  LIN {X -14931.996,Y 2667.355,Z 240.712,A 89.99946,B 0.00000,C 180.00000} ; retreat
  ; Step 2234, bar 855
  LIN {X -14831.996,Y 2667.355,Z 1143.930,A 89.99946,B 0.00000,C 180.00000} ; outside
  LIN {X -14831.996,Y 2667.355,Z 190.712,A 89.99946,B 0.00000,C 180.00000} ; preinsert
  LIN {X -14831.996,Y 2667.355,Z -59.288,A 89.99946,B 0.00000,C 180.00000} ; insert
  LIN {X -14831.996,Y 2667.355,Z -59.288,A 89.99946,B 0.00000,C 180.00000} ; release
  LIN {X -14831.996,Y 2667.355,Z 240.712,A 89.99946,B 0.00000,C 180.00000} ; retreat
  ; Step 2235, bar 853
  LIN {X -14731.996,Y 2667.355,Z 1143.930,A 89.99946,B 0.00000,C 180.00000} ; outside
  LIN {X -14731.996,Y 2667.355,Z 190.712,A 89.99946,B 0.00000,C 180.00000} ; preinsert
  LIN {X -14731.996,Y 2667.355,Z -59.288,A 89.99946,B 0.00000,C 180.00000} ; insert
  LIN {X -14731.996,Y 2667.355,Z -59.288,A 89.99946,B 0.00000,C 180.00000} ; release
  LIN {X -14731.996,Y 2667.355,Z 240.712,A 89.99946,B 0.00000,C 180.00000} ; retreat
  ; Step 2236, bar 851
  LIN {X -14631.996,Y 2667.355,Z 1143.930,A 89.99946,B 0.00000,C 180.00000} ; outside
  LIN {X -14631.996,Y 2667.355,Z 190.712,A 89.99946,B 0.00000,C 180.00000} ; preinsert
  LIN {X -14631.996,Y 2667.355,Z -59.288,A 89.99946,B 0.00000,C 180.00000} ; insert
  LIN {X -14631.996,Y 2667.355,Z -59.288,A 89.99946,B 0.00000,C 180.00000} ; release
  LIN {X -14631.996,Y 2667.355,Z 240.712,A 89.99946,B 0.00000,C 180.00000} ; retreat
  ; Step 2237, bar 849
  LIN {X -14531.996,Y 2667.355,Z 1143.930,A 89.99946,B 0.00000,C 180.00000} ; outside
  LIN {X -14531.996,Y 2667.355,Z 190.712,A 89.99946,B 0.00000,C 180.00000} ; preinsert
  LIN {X -14531.996,Y 2667.355,Z -59.288,A 89.99946,B 0.00000,C 180.00000} ; insert
  LIN {X -14531.996,Y 2667.355,Z -59.288,A 89.99946,B 0.00000,C 180.00000} ; release
  LIN {X -14531.996,Y 2667.355,Z 240.712,A 89.99946,B 0.00000,C 180.00000} ; retreat
  ; Step 2238, bar 847
  LIN {X -14431.996,Y 2667.355,Z 1143.930,A 89.99946,B 0.00000,C 180.00000} ; outside
  LIN {X -14431.996,Y 2667.355,Z 190.712,A 89.99946,B 0.00000,C 180.00000} ; preinsert
  LIN {X -14431.996,Y 2667.355,Z -59.288,A 89.99946,B 0.00000,C 180.00000} ; insert
  LIN {X -14431.996,Y 2667.355,Z -59.288,A 89.99946,B 0.00000,C 180.00000} ; release
  LIN {X -14431.996,Y 2667.355,Z 240.712,A 89.99946,B 0.00000,C 180.00000} ; retreat
  ; Step 2239, bar 845
  LIN {X -14331.996,Y 2667.355,Z 1143.930,A 89.99946,B 0.00000,C 180.00000} ; outside
  LIN {X -14331.996,Y 2667.355,Z 190.712,A 89.99946,B 0.00000,C 180.00000} ; preinsert
  LIN {X -14331.996,Y 2667.355,Z -59.288,A 89.99946,B 0.00000,C 180.00000} ; insert
  LIN {X -14331.996,Y 2667.355,Z -59.288,A 89.99946,B 0.00000,C 180.00000} ; release
  LIN {X -14331.996,Y 2667.355,Z 240.712,A 89.99946,B 0.00000,C 180.00000} ; retreat
  ; Step 2240, bar 843
  LIN {X -14231.996,Y 2667.355,Z 1143.930,A 89.99946,B 0.00000,C 180.00000} ; outside
  LIN {X -14231.996,Y 2667.355,Z 190.712,A 89.99946,B 0.00000,C 180.00000} ; preinsert
  LIN {X -14231.996,Y 2667.355,Z -59.288,A 89.99946,B 0.00000,C 180.00000} ; insert
  LIN {X -14231.996,Y 2667.355,Z -59.288,A 89.99946,B 0.00000,C 180.00000} ; release
  LIN {X -14231.996,Y 2667.355,Z 240.712,A 89.99946,B 0.00000,C 180.00000} ; retreat
  ; Step 2241, bar 841
  LIN {X -14131.996,Y 2667.355,Z 1143.930,A 89.99946,B 0.00000,C 180.00000} ; outside
  LIN {X -14131.996,Y 2667.355,Z 190.712,A 89.99946,B 0.00000,C 180.00000} ; preinsert
  LIN {X -14131.996,Y 2667.355,Z -59.288,A 89.99946,B 0.00000,C 180.00000} ; insert
  LIN {X -14131.996,Y 2667.355,Z -59.288,A 89.99946,B 0.00000,C 180.00000} ; release
  LIN {X -14131.996,Y 2667.355,Z 240.712,A 89.99946,B 0.00000,C 180.00000} ; retreat
  ; Step 2242, bar 839
  LIN {X -13831.996,Y 2667.355,Z 1143.930,A 89.99946,B 0.00000,C 180.00000} ; outside
  LIN {X -13831.996,Y 2667.355,Z 190.712,A 89.99946,B 0.00000,C 180.00000} ; preinsert
  LIN {X -13831.996,Y 2667.355,Z -59.288,A 89.99946,B 0.00000,C 180.00000} ; insert
  LIN {X -13831.996,Y 2667.355,Z -59.288,A 89.99946,B 0.00000,C 180.00000} ; release
  LIN {X -13831.996,Y 2667.355,Z 240.712,A 89.99946,B 0.00000,C 180.00000} ; retreat
  ; Step 2243, bar 837
  LIN {X -13731.996,Y 2667.355,Z 1143.930,A 89.99946,B 0.00000,C 180.00000} ; outside
  LIN {X -13731.996,Y 2667.355,Z 190.712,A 89.99946,B 0.00000,C 180.00000} ; preinsert
  LIN {X -13731.996,Y 2667.355,Z -59.288,A 89.99946,B 0.00000,C 180.00000} ; insert
  LIN {X -13731.996,Y 2667.355,Z -59.288,A 89.99946,B 0.00000,C 180.00000} ; release
  LIN {X -13731.996,Y 2667.355,Z 240.712,A 89.99946,B 0.00000,C 180.00000} ; retreat
  ; Step 2244, bar 835
  LIN {X -13631.996,Y 2667.355,Z 1143.930,A 89.99946,B 0.00000,C 180.00000} ; outside
  LIN {X -13631.996,Y 2667.355,Z 190.712,A 89.99946,B 0.00000,C 180.00000} ; preinsert
  LIN {X -13631.996,Y 2667.355,Z -59.288,A 89.99946,B 0.00000,C 180.00000} ; insert
  LIN {X -13631.996,Y 2667.355,Z -59.288,A 89.99946,B 0.00000,C 180.00000} ; release
  LIN {X -13631.996,Y 2667.355,Z 240.712,A 89.99946,B 0.00000,C 180.00000} ; retreat
  ; Step 2245, bar 833
  LIN {X -13531.996,Y 2667.355,Z 1143.930,A 89.99946,B 0.00000,C 180.00000} ; outside
  LIN {X -13531.996,Y 2667.355,Z 190.712,A 89.99946,B 0.00000,C 180.00000} ; preinsert
  LIN {X -13531.996,Y 2667.355,Z -59.288,A 89.99946,B 0.00000,C 180.00000} ; insert
  LIN {X -13531.996,Y 2667.355,Z -59.288,A 89.99946,B 0.00000,C 180.00000} ; release
  LIN {X -13531.996,Y 2667.355,Z 240.712,A 89.99946,B 0.00000,C 180.00000} ; retreat
  ; Step 2246, bar 831
  LIN {X -13431.996,Y 2667.355,Z 1143.930,A 89.99946,B 0.00000,C 180.00000} ; outside
  LIN {X -13431.996,Y 2667.355,Z 190.712,A 89.99946,B 0.00000,C 180.00000} ; preinsert
  LIN {X -13431.996,Y 2667.355,Z -59.288,A 89.99946,B 0.00000,C 180.00000} ; insert
  LIN {X -13431.996,Y 2667.355,Z -59.288,A 89.99946,B 0.00000,C 180.00000} ; release
  LIN {X -13431.996,Y 2667.355,Z 240.712,A 89.99946,B 0.00000,C 180.00000} ; retreat
  ; Step 2247, bar 829
  LIN {X -13331.996,Y 2667.355,Z 1143.930,A 89.99946,B 0.00000,C 180.00000} ; outside
  LIN {X -13331.996,Y 2667.355,Z 190.712,A 89.99946,B 0.00000,C 180.00000} ; preinsert
  LIN {X -13331.996,Y 2667.355,Z -59.288,A 89.99946,B 0.00000,C 180.00000} ; insert
  LIN {X -13331.996,Y 2667.355,Z -59.288,A 89.99946,B 0.00000,C 180.00000} ; release
  LIN {X -13331.996,Y 2667.355,Z 240.712,A 89.99946,B 0.00000,C 180.00000} ; retreat
  ; Step 2248, bar 827
  LIN {X -13231.996,Y 2667.355,Z 1143.930,A 89.99946,B 0.00000,C 180.00000} ; outside
  LIN {X -13231.996,Y 2667.355,Z 190.712,A 89.99946,B 0.00000,C 180.00000} ; preinsert
  LIN {X -13231.996,Y 2667.355,Z -59.288,A 89.99946,B 0.00000,C 180.00000} ; insert
  LIN {X -13231.996,Y 2667.355,Z -59.288,A 89.99946,B 0.00000,C 180.00000} ; release
  LIN {X -13231.996,Y 2667.355,Z 240.712,A 89.99946,B 0.00000,C 180.00000} ; retreat
  ; Step 2249, bar 825
  LIN {X -13131.996,Y 2667.355,Z 1143.930,A 89.99946,B 0.00000,C 180.00000} ; outside
  LIN {X -13131.996,Y 2667.355,Z 190.712,A 89.99946,B 0.00000,C 180.00000} ; preinsert
  LIN {X -13131.996,Y 2667.355,Z -59.288,A 89.99946,B 0.00000,C 180.00000} ; insert
  LIN {X -13131.996,Y 2667.355,Z -59.288,A 89.99946,B 0.00000,C 180.00000} ; release
  LIN {X -13131.996,Y 2667.355,Z 240.712,A 89.99946,B 0.00000,C 180.00000} ; retreat
  ; Step 2250, bar 823
  LIN {X -13031.996,Y 2667.355,Z 1143.930,A 89.99946,B 0.00000,C 180.00000} ; outside
  LIN {X -13031.996,Y 2667.355,Z 190.712,A 89.99946,B 0.00000,C 180.00000} ; preinsert
  LIN {X -13031.996,Y 2667.355,Z -59.288,A 89.99946,B 0.00000,C 180.00000} ; insert
  LIN {X -13031.996,Y 2667.355,Z -59.288,A 89.99946,B 0.00000,C 180.00000} ; release
  LIN {X -13031.996,Y 2667.355,Z 240.712,A 89.99946,B 0.00000,C 180.00000} ; retreat
  ; Step 2251, bar 821
  LIN {X -12931.996,Y 2667.355,Z 1143.930,A 89.99946,B 0.00000,C 180.00000} ; outside
  LIN {X -12931.996,Y 2667.355,Z 190.712,A 89.99946,B 0.00000,C 180.00000} ; preinsert
  LIN {X -12931.996,Y 2667.355,Z -59.288,A 89.99946,B 0.00000,C 180.00000} ; insert
  LIN {X -12931.996,Y 2667.355,Z -59.288,A 89.99946,B 0.00000,C 180.00000} ; release
  LIN {X -12931.996,Y 2667.355,Z 240.712,A 89.99946,B 0.00000,C 180.00000} ; retreat
  ; Step 2252, bar 819
  LIN {X -12831.996,Y 2667.355,Z 1143.930,A 89.99946,B 0.00000,C 180.00000} ; outside
  LIN {X -12831.996,Y 2667.355,Z 190.712,A 89.99946,B 0.00000,C 180.00000} ; preinsert
  LIN {X -12831.996,Y 2667.355,Z -59.288,A 89.99946,B 0.00000,C 180.00000} ; insert
  LIN {X -12831.996,Y 2667.355,Z -59.288,A 89.99946,B 0.00000,C 180.00000} ; release
  LIN {X -12831.996,Y 2667.355,Z 240.712,A 89.99946,B 0.00000,C 180.00000} ; retreat
  ; Step 2253, bar 817
  LIN {X -12731.996,Y 2667.355,Z 1143.930,A 89.99946,B 0.00000,C 180.00000} ; outside
  LIN {X -12731.996,Y 2667.355,Z 190.712,A 89.99946,B 0.00000,C 180.00000} ; preinsert
  LIN {X -12731.996,Y 2667.355,Z -59.288,A 89.99946,B 0.00000,C 180.00000} ; insert
  LIN {X -12731.996,Y 2667.355,Z -59.288,A 89.99946,B 0.00000,C 180.00000} ; release
  LIN {X -12731.996,Y 2667.355,Z 240.712,A 89.99946,B 0.00000,C 180.00000} ; retreat
  ; Step 2254, bar 815
  LIN {X -12631.996,Y 2667.355,Z 1143.930,A 89.99946,B 0.00000,C 180.00000} ; outside
  LIN {X -12631.996,Y 2667.355,Z 190.712,A 89.99946,B 0.00000,C 180.00000} ; preinsert
  LIN {X -12631.996,Y 2667.355,Z -59.288,A 89.99946,B 0.00000,C 180.00000} ; insert
  LIN {X -12631.996,Y 2667.355,Z -59.288,A 89.99946,B 0.00000,C 180.00000} ; release
  LIN {X -12631.996,Y 2667.355,Z 240.712,A 89.99946,B 0.00000,C 180.00000} ; retreat
  ; Step 2255, bar 813
  LIN {X -12531.996,Y 2667.355,Z 1143.930,A 89.99946,B 0.00000,C 180.00000} ; outside
  LIN {X -12531.996,Y 2667.355,Z 190.712,A 89.99946,B 0.00000,C 180.00000} ; preinsert
  LIN {X -12531.996,Y 2667.355,Z -59.288,A 89.99946,B 0.00000,C 180.00000} ; insert
  LIN {X -12531.996,Y 2667.355,Z -59.288,A 89.99946,B 0.00000,C 180.00000} ; release
  LIN {X -12531.996,Y 2667.355,Z 240.712,A 89.99946,B 0.00000,C 180.00000} ; retreat
  ; Step 2256, bar 811
  LIN {X -12431.996,Y 2667.355,Z 1143.930,A 89.99946,B 0.00000,C 180.00000} ; outside
  LIN {X -12431.996,Y 2667.355,Z 190.712,A 89.99946,B 0.00000,C 180.00000} ; preinsert
  LIN {X -12431.996,Y 2667.355,Z -59.288,A 89.99946,B 0.00000,C 180.00000} ; insert
  LIN {X -12431.996,Y 2667.355,Z -59.288,A 89.99946,B 0.00000,C 180.00000} ; release
  LIN {X -12431.996,Y 2667.355,Z 240.712,A 89.99946,B 0.00000,C 180.00000} ; retreat
  ; Step 2257, bar 809
  LIN {X -12331.996,Y 2667.355,Z 1143.930,A 89.99946,B 0.00000,C 180.00000} ; outside
  LIN {X -12331.996,Y 2667.355,Z 190.712,A 89.99946,B 0.00000,C 180.00000} ; preinsert
  LIN {X -12331.996,Y 2667.355,Z -59.288,A 89.99946,B 0.00000,C 180.00000} ; insert
  LIN {X -12331.996,Y 2667.355,Z -59.288,A 89.99946,B 0.00000,C 180.00000} ; release
  LIN {X -12331.996,Y 2667.355,Z 240.712,A 89.99946,B 0.00000,C 180.00000} ; retreat
  ; Step 2258, bar 807
  LIN {X -12231.996,Y 2667.355,Z 1143.930,A 89.99946,B 0.00000,C 180.00000} ; outside
  LIN {X -12231.996,Y 2667.355,Z 190.712,A 89.99946,B 0.00000,C 180.00000} ; preinsert
  LIN {X -12231.996,Y 2667.355,Z -59.288,A 89.99946,B 0.00000,C 180.00000} ; insert
  LIN {X -12231.996,Y 2667.355,Z -59.288,A 89.99946,B 0.00000,C 180.00000} ; release
  LIN {X -12231.996,Y 2667.355,Z 240.712,A 89.99946,B 0.00000,C 180.00000} ; retreat
  ; Step 2259, bar 805
  LIN {X -12106.996,Y 2667.355,Z 1143.930,A 89.99946,B 0.00000,C 180.00000} ; outside
  LIN {X -12106.996,Y 2667.355,Z 190.712,A 89.99946,B 0.00000,C 180.00000} ; preinsert
  LIN {X -12106.996,Y 2667.355,Z -59.288,A 89.99946,B 0.00000,C 180.00000} ; insert
  LIN {X -12106.996,Y 2667.355,Z -59.288,A 89.99946,B 0.00000,C 180.00000} ; release
  LIN {X -12106.996,Y 2667.355,Z 240.712,A 89.99946,B 0.00000,C 180.00000} ; retreat
  ; Step 2260, bar 803
  LIN {X -11981.996,Y 2667.355,Z 1143.930,A 89.99946,B 0.00000,C 180.00000} ; outside
  LIN {X -11981.996,Y 2667.355,Z 190.712,A 89.99946,B 0.00000,C 180.00000} ; preinsert
  LIN {X -11981.996,Y 2667.355,Z -59.288,A 89.99946,B 0.00000,C 180.00000} ; insert
  LIN {X -11981.996,Y 2667.355,Z -59.288,A 89.99946,B 0.00000,C 180.00000} ; release
  LIN {X -11981.996,Y 2667.355,Z 240.712,A 89.99946,B 0.00000,C 180.00000} ; retreat
  ; Step 2261, bar 801
  LIN {X -11856.996,Y 2667.355,Z 1143.930,A 89.99946,B 0.00000,C 180.00000} ; outside
  LIN {X -11856.996,Y 2667.355,Z 190.712,A 89.99946,B 0.00000,C 180.00000} ; preinsert
  LIN {X -11856.996,Y 2667.355,Z -59.288,A 89.99946,B 0.00000,C 180.00000} ; insert
  LIN {X -11856.996,Y 2667.355,Z -59.288,A 89.99946,B 0.00000,C 180.00000} ; release
  LIN {X -11856.996,Y 2667.355,Z 240.712,A 89.99946,B 0.00000,C 180.00000} ; retreat
  ; Step 2262, bar 799
  LIN {X -11731.996,Y 2667.355,Z 1143.930,A 89.99946,B 0.00000,C 180.00000} ; outside
  LIN {X -11731.996,Y 2667.355,Z 190.712,A 89.99946,B 0.00000,C 180.00000} ; preinsert
  LIN {X -11731.996,Y 2667.355,Z -59.288,A 89.99946,B 0.00000,C 180.00000} ; insert
  LIN {X -11731.996,Y 2667.355,Z -59.288,A 89.99946,B 0.00000,C 180.00000} ; release
  LIN {X -11731.996,Y 2667.355,Z 240.712,A 89.99946,B 0.00000,C 180.00000} ; retreat
  ; Step 2263, bar 797
  LIN {X -11606.996,Y 2667.355,Z 1143.930,A 89.99946,B 0.00000,C 180.00000} ; outside
  LIN {X -11606.996,Y 2667.355,Z 190.712,A 89.99946,B 0.00000,C 180.00000} ; preinsert
  LIN {X -11606.996,Y 2667.355,Z -59.288,A 89.99946,B 0.00000,C 180.00000} ; insert
  LIN {X -11606.996,Y 2667.355,Z -59.288,A 89.99946,B 0.00000,C 180.00000} ; release
  LIN {X -11606.996,Y 2667.355,Z 240.712,A 89.99946,B 0.00000,C 180.00000} ; retreat
  ; Step 2264, bar 795
  LIN {X -11481.996,Y 2667.355,Z 1143.930,A 89.99946,B 0.00000,C 180.00000} ; outside
  LIN {X -11481.996,Y 2667.355,Z 190.712,A 89.99946,B 0.00000,C 180.00000} ; preinsert
  LIN {X -11481.996,Y 2667.355,Z -59.288,A 89.99946,B 0.00000,C 180.00000} ; insert
  LIN {X -11481.996,Y 2667.355,Z -59.288,A 89.99946,B 0.00000,C 180.00000} ; release
  LIN {X -11481.996,Y 2667.355,Z 240.712,A 89.99946,B 0.00000,C 180.00000} ; retreat
  ; Step 2265, bar 793
  LIN {X -11356.996,Y 2667.355,Z 1143.930,A 89.99946,B 0.00000,C 180.00000} ; outside
  LIN {X -11356.996,Y 2667.355,Z 190.712,A 89.99946,B 0.00000,C 180.00000} ; preinsert
  LIN {X -11356.996,Y 2667.355,Z -59.288,A 89.99946,B 0.00000,C 180.00000} ; insert
  LIN {X -11356.996,Y 2667.355,Z -59.288,A 89.99946,B 0.00000,C 180.00000} ; release
  LIN {X -11356.996,Y 2667.355,Z 240.712,A 89.99946,B 0.00000,C 180.00000} ; retreat
  ; Step 2266, bar 791
  LIN {X -11231.996,Y 2667.355,Z 1143.930,A 89.99946,B 0.00000,C 180.00000} ; outside
  LIN {X -11231.996,Y 2667.355,Z 190.712,A 89.99946,B 0.00000,C 180.00000} ; preinsert
  LIN {X -11231.996,Y 2667.355,Z -59.288,A 89.99946,B 0.00000,C 180.00000} ; insert
  LIN {X -11231.996,Y 2667.355,Z -59.288,A 89.99946,B 0.00000,C 180.00000} ; release
  LIN {X -11231.996,Y 2667.355,Z 240.712,A 89.99946,B 0.00000,C 180.00000} ; retreat
  ; Step 2267, bar 789
  LIN {X -11106.996,Y 2667.355,Z 1143.930,A 89.99946,B 0.00000,C 180.00000} ; outside
  LIN {X -11106.996,Y 2667.355,Z 190.712,A 89.99946,B 0.00000,C 180.00000} ; preinsert
  LIN {X -11106.996,Y 2667.355,Z -59.288,A 89.99946,B 0.00000,C 180.00000} ; insert
  LIN {X -11106.996,Y 2667.355,Z -59.288,A 89.99946,B 0.00000,C 180.00000} ; release
  LIN {X -11106.996,Y 2667.355,Z 240.712,A 89.99946,B 0.00000,C 180.00000} ; retreat
  ; Step 2268, bar 787
  LIN {X -10981.996,Y 2667.355,Z 1143.930,A 89.99946,B 0.00000,C 180.00000} ; outside
  LIN {X -10981.996,Y 2667.355,Z 190.712,A 89.99946,B 0.00000,C 180.00000} ; preinsert
  LIN {X -10981.996,Y 2667.355,Z -59.288,A 89.99946,B 0.00000,C 180.00000} ; insert
  LIN {X -10981.996,Y 2667.355,Z -59.288,A 89.99946,B 0.00000,C 180.00000} ; release
  LIN {X -10981.996,Y 2667.355,Z 240.712,A 89.99946,B 0.00000,C 180.00000} ; retreat
  ; Step 2269, bar 785
  LIN {X -10856.996,Y 2667.355,Z 1143.930,A 89.99946,B 0.00000,C 180.00000} ; outside
  LIN {X -10856.996,Y 2667.355,Z 190.712,A 89.99946,B 0.00000,C 180.00000} ; preinsert
  LIN {X -10856.996,Y 2667.355,Z -59.288,A 89.99946,B 0.00000,C 180.00000} ; insert
  LIN {X -10856.996,Y 2667.355,Z -59.288,A 89.99946,B 0.00000,C 180.00000} ; release
  LIN {X -10856.996,Y 2667.355,Z 240.712,A 89.99946,B 0.00000,C 180.00000} ; retreat
  ; Step 2270, bar 783
  LIN {X -10731.996,Y 2667.355,Z 1143.930,A 89.99946,B 0.00000,C 180.00000} ; outside
  LIN {X -10731.996,Y 2667.355,Z 190.712,A 89.99946,B 0.00000,C 180.00000} ; preinsert
  LIN {X -10731.996,Y 2667.355,Z -59.288,A 89.99946,B 0.00000,C 180.00000} ; insert
  LIN {X -10731.996,Y 2667.355,Z -59.288,A 89.99946,B 0.00000,C 180.00000} ; release
  LIN {X -10731.996,Y 2667.355,Z 240.712,A 89.99946,B 0.00000,C 180.00000} ; retreat
  ; Step 2271, bar 781
  LIN {X -10606.996,Y 2667.355,Z 1143.930,A 89.99946,B 0.00000,C 180.00000} ; outside
  LIN {X -10606.996,Y 2667.355,Z 190.712,A 89.99946,B 0.00000,C 180.00000} ; preinsert
  LIN {X -10606.996,Y 2667.355,Z -59.288,A 89.99946,B 0.00000,C 180.00000} ; insert
  LIN {X -10606.996,Y 2667.355,Z -59.288,A 89.99946,B 0.00000,C 180.00000} ; release
  LIN {X -10606.996,Y 2667.355,Z 240.712,A 89.99946,B 0.00000,C 180.00000} ; retreat
  ; Step 2272, bar 779
  LIN {X -10481.996,Y 2667.355,Z 1143.930,A 89.99946,B 0.00000,C 180.00000} ; outside
  LIN {X -10481.996,Y 2667.355,Z 190.712,A 89.99946,B 0.00000,C 180.00000} ; preinsert
  LIN {X -10481.996,Y 2667.355,Z -59.288,A 89.99946,B 0.00000,C 180.00000} ; insert
  LIN {X -10481.996,Y 2667.355,Z -59.288,A 89.99946,B 0.00000,C 180.00000} ; release
  LIN {X -10481.996,Y 2667.355,Z 240.712,A 89.99946,B 0.00000,C 180.00000} ; retreat
  ; Step 2273, bar 777
  LIN {X -10356.996,Y 2667.355,Z 1143.930,A 89.99946,B 0.00000,C 180.00000} ; outside
  LIN {X -10356.996,Y 2667.355,Z 190.712,A 89.99946,B 0.00000,C 180.00000} ; preinsert
  LIN {X -10356.996,Y 2667.355,Z -59.288,A 89.99946,B 0.00000,C 180.00000} ; insert
  LIN {X -10356.996,Y 2667.355,Z -59.288,A 89.99946,B 0.00000,C 180.00000} ; release
  LIN {X -10356.996,Y 2667.355,Z 240.712,A 89.99946,B 0.00000,C 180.00000} ; retreat
  ; Step 2274, bar 775
  LIN {X -10231.996,Y 2667.355,Z 1143.930,A 89.99946,B 0.00000,C 180.00000} ; outside
  LIN {X -10231.996,Y 2667.355,Z 190.712,A 89.99946,B 0.00000,C 180.00000} ; preinsert
  LIN {X -10231.996,Y 2667.355,Z -59.288,A 89.99946,B 0.00000,C 180.00000} ; insert
  LIN {X -10231.996,Y 2667.355,Z -59.288,A 89.99946,B 0.00000,C 180.00000} ; release
  LIN {X -10231.996,Y 2667.355,Z 240.712,A 89.99946,B 0.00000,C 180.00000} ; retreat
  ; Step 2275, bar 773
  LIN {X -10106.996,Y 2667.355,Z 1143.930,A 89.99946,B 0.00000,C 180.00000} ; outside
  LIN {X -10106.996,Y 2667.355,Z 190.712,A 89.99946,B 0.00000,C 180.00000} ; preinsert
  LIN {X -10106.996,Y 2667.355,Z -59.288,A 89.99946,B 0.00000,C 180.00000} ; insert
  LIN {X -10106.996,Y 2667.355,Z -59.288,A 89.99946,B 0.00000,C 180.00000} ; release
  LIN {X -10106.996,Y 2667.355,Z 240.712,A 89.99946,B 0.00000,C 180.00000} ; retreat
  ; Step 2276, bar 771
  LIN {X -9856.996,Y 2667.355,Z 1143.930,A 89.99946,B 0.00000,C 180.00000} ; outside
  LIN {X -9856.996,Y 2667.355,Z 190.712,A 89.99946,B 0.00000,C 180.00000} ; preinsert
  LIN {X -9856.996,Y 2667.355,Z -59.288,A 89.99946,B 0.00000,C 180.00000} ; insert
  LIN {X -9856.996,Y 2667.355,Z -59.288,A 89.99946,B 0.00000,C 180.00000} ; release
  LIN {X -9856.996,Y 2667.355,Z 240.712,A 89.99946,B 0.00000,C 180.00000} ; retreat
  ; Step 2277, bar 769
  LIN {X -9731.996,Y 2667.355,Z 1143.930,A 89.99946,B 0.00000,C 180.00000} ; outside
  LIN {X -9731.996,Y 2667.355,Z 190.712,A 89.99946,B 0.00000,C 180.00000} ; preinsert
  LIN {X -9731.996,Y 2667.355,Z -59.288,A 89.99946,B 0.00000,C 180.00000} ; insert
  LIN {X -9731.996,Y 2667.355,Z -59.288,A 89.99946,B 0.00000,C 180.00000} ; release
  LIN {X -9731.996,Y 2667.355,Z 240.712,A 89.99946,B 0.00000,C 180.00000} ; retreat
  ; Step 2278, bar 767
  LIN {X -9606.996,Y 2667.355,Z 1143.930,A 89.99946,B 0.00000,C 180.00000} ; outside
  LIN {X -9606.996,Y 2667.355,Z 190.712,A 89.99946,B 0.00000,C 180.00000} ; preinsert
  LIN {X -9606.996,Y 2667.355,Z -59.288,A 89.99946,B 0.00000,C 180.00000} ; insert
  LIN {X -9606.996,Y 2667.355,Z -59.288,A 89.99946,B 0.00000,C 180.00000} ; release
  LIN {X -9606.996,Y 2667.355,Z 240.712,A 89.99946,B 0.00000,C 180.00000} ; retreat
  ; Step 2279, bar 765
  LIN {X -9481.996,Y 2667.355,Z 1143.930,A 89.99946,B 0.00000,C 180.00000} ; outside
  LIN {X -9481.996,Y 2667.355,Z 190.712,A 89.99946,B 0.00000,C 180.00000} ; preinsert
  LIN {X -9481.996,Y 2667.355,Z -59.288,A 89.99946,B 0.00000,C 180.00000} ; insert
  LIN {X -9481.996,Y 2667.355,Z -59.288,A 89.99946,B 0.00000,C 180.00000} ; release
  LIN {X -9481.996,Y 2667.355,Z 240.712,A 89.99946,B 0.00000,C 180.00000} ; retreat
  ; Step 2280, bar 763
  LIN {X -9356.996,Y 2667.355,Z 1143.930,A 89.99946,B 0.00000,C 180.00000} ; outside
  LIN {X -9356.996,Y 2667.355,Z 190.712,A 89.99946,B 0.00000,C 180.00000} ; preinsert
  LIN {X -9356.996,Y 2667.355,Z -59.288,A 89.99946,B 0.00000,C 180.00000} ; insert
  LIN {X -9356.996,Y 2667.355,Z -59.288,A 89.99946,B 0.00000,C 180.00000} ; release
  LIN {X -9356.996,Y 2667.355,Z 240.712,A 89.99946,B 0.00000,C 180.00000} ; retreat
  ; Step 2281, bar 761
  LIN {X -9231.996,Y 2667.355,Z 1143.930,A 89.99946,B 0.00000,C 180.00000} ; outside
  LIN {X -9231.996,Y 2667.355,Z 190.712,A 89.99946,B 0.00000,C 180.00000} ; preinsert
  LIN {X -9231.996,Y 2667.355,Z -59.288,A 89.99946,B 0.00000,C 180.00000} ; insert
  LIN {X -9231.996,Y 2667.355,Z -59.288,A 89.99946,B 0.00000,C 180.00000} ; release
  LIN {X -9231.996,Y 2667.355,Z 240.712,A 89.99946,B 0.00000,C 180.00000} ; retreat
  ; Step 2282, bar 759
  LIN {X -9106.996,Y 2667.355,Z 1143.930,A 89.99946,B 0.00000,C 180.00000} ; outside
  LIN {X -9106.996,Y 2667.355,Z 190.712,A 89.99946,B 0.00000,C 180.00000} ; preinsert
  LIN {X -9106.996,Y 2667.355,Z -59.288,A 89.99946,B 0.00000,C 180.00000} ; insert
  LIN {X -9106.996,Y 2667.355,Z -59.288,A 89.99946,B 0.00000,C 180.00000} ; release
  LIN {X -9106.996,Y 2667.355,Z 240.712,A 89.99946,B 0.00000,C 180.00000} ; retreat
  ; Step 2283, bar 757
  LIN {X -8981.996,Y 2667.355,Z 1143.930,A 89.99946,B 0.00000,C 180.00000} ; outside
  LIN {X -8981.996,Y 2667.355,Z 190.712,A 89.99946,B 0.00000,C 180.00000} ; preinsert
  LIN {X -8981.996,Y 2667.355,Z -59.288,A 89.99946,B 0.00000,C 180.00000} ; insert
  LIN {X -8981.996,Y 2667.355,Z -59.288,A 89.99946,B 0.00000,C 180.00000} ; release
  LIN {X -8981.996,Y 2667.355,Z 240.712,A 89.99946,B 0.00000,C 180.00000} ; retreat
  ; Step 2284, bar 755
  LIN {X -8856.996,Y 2667.355,Z 1143.930,A 89.99946,B 0.00000,C 180.00000} ; outside
  LIN {X -8856.996,Y 2667.355,Z 190.712,A 89.99946,B 0.00000,C 180.00000} ; preinsert
  LIN {X -8856.996,Y 2667.355,Z -59.288,A 89.99946,B 0.00000,C 180.00000} ; insert
  LIN {X -8856.996,Y 2667.355,Z -59.288,A 89.99946,B 0.00000,C 180.00000} ; release
  LIN {X -8856.996,Y 2667.355,Z 240.712,A 89.99946,B 0.00000,C 180.00000} ; retreat
  ; Step 2285, bar 753
  LIN {X -8731.996,Y 2667.355,Z 1143.930,A 89.99946,B 0.00000,C 180.00000} ; outside
  LIN {X -8731.996,Y 2667.355,Z 190.712,A 89.99946,B 0.00000,C 180.00000} ; preinsert
  LIN {X -8731.996,Y 2667.355,Z -59.288,A 89.99946,B 0.00000,C 180.00000} ; insert
  LIN {X -8731.996,Y 2667.355,Z -59.288,A 89.99946,B 0.00000,C 180.00000} ; release
  LIN {X -8731.996,Y 2667.355,Z 240.712,A 89.99946,B 0.00000,C 180.00000} ; retreat
  ; Step 2286, bar 751
  LIN {X -8606.996,Y 2667.355,Z 1143.930,A 89.99946,B 0.00000,C 180.00000} ; outside
  LIN {X -8606.996,Y 2667.355,Z 190.712,A 89.99946,B 0.00000,C 180.00000} ; preinsert
  LIN {X -8606.996,Y 2667.355,Z -59.288,A 89.99946,B 0.00000,C 180.00000} ; insert
  LIN {X -8606.996,Y 2667.355,Z -59.288,A 89.99946,B 0.00000,C 180.00000} ; release
  LIN {X -8606.996,Y 2667.355,Z 240.712,A 89.99946,B 0.00000,C 180.00000} ; retreat
  ; Step 2287, bar 749
  LIN {X -8481.996,Y 2667.355,Z 1143.930,A 89.99946,B 0.00000,C 180.00000} ; outside
  LIN {X -8481.996,Y 2667.355,Z 190.712,A 89.99946,B 0.00000,C 180.00000} ; preinsert
  LIN {X -8481.996,Y 2667.355,Z -59.288,A 89.99946,B 0.00000,C 180.00000} ; insert
  LIN {X -8481.996,Y 2667.355,Z -59.288,A 89.99946,B 0.00000,C 180.00000} ; release
  LIN {X -8481.996,Y 2667.355,Z 240.712,A 89.99946,B 0.00000,C 180.00000} ; retreat
  ; Step 2288, bar 747
  LIN {X -8356.996,Y 2667.355,Z 1143.930,A 89.99946,B 0.00000,C 180.00000} ; outside
  LIN {X -8356.996,Y 2667.355,Z 190.712,A 89.99946,B 0.00000,C 180.00000} ; preinsert
  LIN {X -8356.996,Y 2667.355,Z -59.288,A 89.99946,B 0.00000,C 180.00000} ; insert
  LIN {X -8356.996,Y 2667.355,Z -59.288,A 89.99946,B 0.00000,C 180.00000} ; release
  LIN {X -8356.996,Y 2667.355,Z 240.712,A 89.99946,B 0.00000,C 180.00000} ; retreat
  ; Step 2289, bar 745
  LIN {X -8231.996,Y 2667.355,Z 1143.930,A 89.99946,B 0.00000,C 180.00000} ; outside
  LIN {X -8231.996,Y 2667.355,Z 190.712,A 89.99946,B 0.00000,C 180.00000} ; preinsert
  LIN {X -8231.996,Y 2667.355,Z -59.288,A 89.99946,B 0.00000,C 180.00000} ; insert
  LIN {X -8231.996,Y 2667.355,Z -59.288,A 89.99946,B 0.00000,C 180.00000} ; release
  LIN {X -8231.996,Y 2667.355,Z 240.712,A 89.99946,B 0.00000,C 180.00000} ; retreat
  ; Step 2290, bar 743
  LIN {X -8106.996,Y 2667.355,Z 1143.930,A 89.99946,B 0.00000,C 180.00000} ; outside
  LIN {X -8106.996,Y 2667.355,Z 190.712,A 89.99946,B 0.00000,C 180.00000} ; preinsert
  LIN {X -8106.996,Y 2667.355,Z -59.288,A 89.99946,B 0.00000,C 180.00000} ; insert
  LIN {X -8106.996,Y 2667.355,Z -59.288,A 89.99946,B 0.00000,C 180.00000} ; release
  LIN {X -8106.996,Y 2667.355,Z 240.712,A 89.99946,B 0.00000,C 180.00000} ; retreat
  ; Step 2291, bar 741
  LIN {X -7981.996,Y 2667.355,Z 1143.930,A 89.99946,B 0.00000,C 180.00000} ; outside
  LIN {X -7981.996,Y 2667.355,Z 190.712,A 89.99946,B 0.00000,C 180.00000} ; preinsert
  LIN {X -7981.996,Y 2667.355,Z -59.288,A 89.99946,B 0.00000,C 180.00000} ; insert
  LIN {X -7981.996,Y 2667.355,Z -59.288,A 89.99946,B 0.00000,C 180.00000} ; release
  LIN {X -7981.996,Y 2667.355,Z 240.712,A 89.99946,B 0.00000,C 180.00000} ; retreat
  ; Step 2292, bar 739
  LIN {X -7856.996,Y 2667.355,Z 1143.930,A 89.99946,B 0.00000,C 180.00000} ; outside
  LIN {X -7856.996,Y 2667.355,Z 190.712,A 89.99946,B 0.00000,C 180.00000} ; preinsert
  LIN {X -7856.996,Y 2667.355,Z -59.288,A 89.99946,B 0.00000,C 180.00000} ; insert
  LIN {X -7856.996,Y 2667.355,Z -59.288,A 89.99946,B 0.00000,C 180.00000} ; release
  LIN {X -7856.996,Y 2667.355,Z 240.712,A 89.99946,B 0.00000,C 180.00000} ; retreat
  ; Step 2293, bar 737
  LIN {X -7731.996,Y 2667.355,Z 1143.930,A 89.99946,B 0.00000,C 180.00000} ; outside
  LIN {X -7731.996,Y 2667.355,Z 190.712,A 89.99946,B 0.00000,C 180.00000} ; preinsert
  LIN {X -7731.996,Y 2667.355,Z -59.288,A 89.99946,B 0.00000,C 180.00000} ; insert
  LIN {X -7731.996,Y 2667.355,Z -59.288,A 89.99946,B 0.00000,C 180.00000} ; release
  LIN {X -7731.996,Y 2667.355,Z 240.712,A 89.99946,B 0.00000,C 180.00000} ; retreat
  ; Step 2294, bar 735
  LIN {X -7606.996,Y 2667.355,Z 1143.930,A 89.99946,B 0.00000,C 180.00000} ; outside
  LIN {X -7606.996,Y 2667.355,Z 190.712,A 89.99946,B 0.00000,C 180.00000} ; preinsert
  LIN {X -7606.996,Y 2667.355,Z -59.288,A 89.99946,B 0.00000,C 180.00000} ; insert
  LIN {X -7606.996,Y 2667.355,Z -59.288,A 89.99946,B 0.00000,C 180.00000} ; release
  LIN {X -7606.996,Y 2667.355,Z 240.712,A 89.99946,B 0.00000,C 180.00000} ; retreat
  ; Step 2295, bar 733
  LIN {X -7481.996,Y 2667.355,Z 1143.930,A 89.99946,B 0.00000,C 180.00000} ; outside
  LIN {X -7481.996,Y 2667.355,Z 190.712,A 89.99946,B 0.00000,C 180.00000} ; preinsert
  LIN {X -7481.996,Y 2667.355,Z -59.288,A 89.99946,B 0.00000,C 180.00000} ; insert
  LIN {X -7481.996,Y 2667.355,Z -59.288,A 89.99946,B 0.00000,C 180.00000} ; release
  LIN {X -7481.996,Y 2667.355,Z 240.712,A 89.99946,B 0.00000,C 180.00000} ; retreat
  ; Step 2296, bar 731
  LIN {X -7356.996,Y 2667.355,Z 1143.930,A 89.99946,B 0.00000,C 180.00000} ; outside
  LIN {X -7356.996,Y 2667.355,Z 190.712,A 89.99946,B 0.00000,C 180.00000} ; preinsert
  LIN {X -7356.996,Y 2667.355,Z -59.288,A 89.99946,B 0.00000,C 180.00000} ; insert
  LIN {X -7356.996,Y 2667.355,Z -59.288,A 89.99946,B 0.00000,C 180.00000} ; release
  LIN {X -7356.996,Y 2667.355,Z 240.712,A 89.99946,B 0.00000,C 180.00000} ; retreat
  ; Step 2297, bar 729
  LIN {X -7231.996,Y 2667.355,Z 1143.930,A 89.99946,B 0.00000,C 180.00000} ; outside
  LIN {X -7231.996,Y 2667.355,Z 190.712,A 89.99946,B 0.00000,C 180.00000} ; preinsert
  LIN {X -7231.996,Y 2667.355,Z -59.288,A 89.99946,B 0.00000,C 180.00000} ; insert
  LIN {X -7231.996,Y 2667.355,Z -59.288,A 89.99946,B 0.00000,C 180.00000} ; release
  LIN {X -7231.996,Y 2667.355,Z 240.712,A 89.99946,B 0.00000,C 180.00000} ; retreat
  ; Step 2298, bar 727
  LIN {X -7106.996,Y 2667.355,Z 1143.930,A 89.99946,B 0.00000,C 180.00000} ; outside
  LIN {X -7106.996,Y 2667.355,Z 190.712,A 89.99946,B 0.00000,C 180.00000} ; preinsert
  LIN {X -7106.996,Y 2667.355,Z -59.288,A 89.99946,B 0.00000,C 180.00000} ; insert
  LIN {X -7106.996,Y 2667.355,Z -59.288,A 89.99946,B 0.00000,C 180.00000} ; release
  LIN {X -7106.996,Y 2667.355,Z 240.712,A 89.99946,B 0.00000,C 180.00000} ; retreat
  ; Step 2299, bar 725
  LIN {X -6981.996,Y 2667.355,Z 1143.930,A 89.99946,B 0.00000,C 180.00000} ; outside
  LIN {X -6981.996,Y 2667.355,Z 190.712,A 89.99946,B 0.00000,C 180.00000} ; preinsert
  LIN {X -6981.996,Y 2667.355,Z -59.288,A 89.99946,B 0.00000,C 180.00000} ; insert
  LIN {X -6981.996,Y 2667.355,Z -59.288,A 89.99946,B 0.00000,C 180.00000} ; release
  LIN {X -6981.996,Y 2667.355,Z 240.712,A 89.99946,B 0.00000,C 180.00000} ; retreat
  ; Step 2300, bar 723
  LIN {X -6856.996,Y 2667.355,Z 1143.930,A 89.99946,B 0.00000,C 180.00000} ; outside
  LIN {X -6856.996,Y 2667.355,Z 190.712,A 89.99946,B 0.00000,C 180.00000} ; preinsert
  LIN {X -6856.996,Y 2667.355,Z -59.288,A 89.99946,B 0.00000,C 180.00000} ; insert
  LIN {X -6856.996,Y 2667.355,Z -59.288,A 89.99946,B 0.00000,C 180.00000} ; release
  LIN {X -6856.996,Y 2667.355,Z 240.712,A 89.99946,B 0.00000,C 180.00000} ; retreat
  ; Step 2301, bar 721
  LIN {X -6731.996,Y 2667.355,Z 1143.930,A 89.99946,B 0.00000,C 180.00000} ; outside
  LIN {X -6731.996,Y 2667.355,Z 190.712,A 89.99946,B 0.00000,C 180.00000} ; preinsert
  LIN {X -6731.996,Y 2667.355,Z -59.288,A 89.99946,B 0.00000,C 180.00000} ; insert
  LIN {X -6731.996,Y 2667.355,Z -59.288,A 89.99946,B 0.00000,C 180.00000} ; release
  LIN {X -6731.996,Y 2667.355,Z 240.712,A 89.99946,B 0.00000,C 180.00000} ; retreat
  ; Step 2302, bar 719
  LIN {X -6606.996,Y 2667.355,Z 1143.930,A 89.99946,B 0.00000,C 180.00000} ; outside
  LIN {X -6606.996,Y 2667.355,Z 190.712,A 89.99946,B 0.00000,C 180.00000} ; preinsert
  LIN {X -6606.996,Y 2667.355,Z -59.288,A 89.99946,B 0.00000,C 180.00000} ; insert
  LIN {X -6606.996,Y 2667.355,Z -59.288,A 89.99946,B 0.00000,C 180.00000} ; release
  LIN {X -6606.996,Y 2667.355,Z 240.712,A 89.99946,B 0.00000,C 180.00000} ; retreat
  ; Step 2303, bar 717
  LIN {X -6481.996,Y 2667.355,Z 1143.930,A 89.99946,B 0.00000,C 180.00000} ; outside
  LIN {X -6481.996,Y 2667.355,Z 190.712,A 89.99946,B 0.00000,C 180.00000} ; preinsert
  LIN {X -6481.996,Y 2667.355,Z -59.288,A 89.99946,B 0.00000,C 180.00000} ; insert
  LIN {X -6481.996,Y 2667.355,Z -59.288,A 89.99946,B 0.00000,C 180.00000} ; release
  LIN {X -6481.996,Y 2667.355,Z 240.712,A 89.99946,B 0.00000,C 180.00000} ; retreat
  ; Step 2304, bar 715
  LIN {X -6356.996,Y 2667.355,Z 1143.930,A 89.99946,B 0.00000,C 180.00000} ; outside
  LIN {X -6356.996,Y 2667.355,Z 190.712,A 89.99946,B 0.00000,C 180.00000} ; preinsert
  LIN {X -6356.996,Y 2667.355,Z -59.288,A 89.99946,B 0.00000,C 180.00000} ; insert
  LIN {X -6356.996,Y 2667.355,Z -59.288,A 89.99946,B 0.00000,C 180.00000} ; release
  LIN {X -6356.996,Y 2667.355,Z 240.712,A 89.99946,B 0.00000,C 180.00000} ; retreat
  ; Step 2305, bar 713
  LIN {X -6231.996,Y 2667.355,Z 1143.930,A 89.99946,B 0.00000,C 180.00000} ; outside
  LIN {X -6231.996,Y 2667.355,Z 190.712,A 89.99946,B 0.00000,C 180.00000} ; preinsert
  LIN {X -6231.996,Y 2667.355,Z -59.288,A 89.99946,B 0.00000,C 180.00000} ; insert
  LIN {X -6231.996,Y 2667.355,Z -59.288,A 89.99946,B 0.00000,C 180.00000} ; release
  LIN {X -6231.996,Y 2667.355,Z 240.712,A 89.99946,B 0.00000,C 180.00000} ; retreat
  ; Step 2306, bar 711
  LIN {X -6106.996,Y 2667.355,Z 1143.930,A 89.99946,B 0.00000,C 180.00000} ; outside
  LIN {X -6106.996,Y 2667.355,Z 190.712,A 89.99946,B 0.00000,C 180.00000} ; preinsert
  LIN {X -6106.996,Y 2667.355,Z -59.288,A 89.99946,B 0.00000,C 180.00000} ; insert
  LIN {X -6106.996,Y 2667.355,Z -59.288,A 89.99946,B 0.00000,C 180.00000} ; release
  LIN {X -6106.996,Y 2667.355,Z 240.712,A 89.99946,B 0.00000,C 180.00000} ; retreat
  ; Step 2307, bar 709
  LIN {X -5856.996,Y 2667.355,Z 1143.930,A 89.99946,B 0.00000,C 180.00000} ; outside
  LIN {X -5856.996,Y 2667.355,Z 190.712,A 89.99946,B 0.00000,C 180.00000} ; preinsert
  LIN {X -5856.996,Y 2667.355,Z -59.288,A 89.99946,B 0.00000,C 180.00000} ; insert
  LIN {X -5856.996,Y 2667.355,Z -59.288,A 89.99946,B 0.00000,C 180.00000} ; release
  LIN {X -5856.996,Y 2667.355,Z 240.712,A 89.99946,B 0.00000,C 180.00000} ; retreat
  ; Step 2308, bar 707
  LIN {X -5731.996,Y 2667.355,Z 1143.930,A 89.99946,B 0.00000,C 180.00000} ; outside
  LIN {X -5731.996,Y 2667.355,Z 190.712,A 89.99946,B 0.00000,C 180.00000} ; preinsert
  LIN {X -5731.996,Y 2667.355,Z -59.288,A 89.99946,B 0.00000,C 180.00000} ; insert
  LIN {X -5731.996,Y 2667.355,Z -59.288,A 89.99946,B 0.00000,C 180.00000} ; release
  LIN {X -5731.996,Y 2667.355,Z 240.712,A 89.99946,B 0.00000,C 180.00000} ; retreat
  ; Step 2309, bar 705
  LIN {X -5606.996,Y 2667.355,Z 1143.930,A 89.99946,B 0.00000,C 180.00000} ; outside
  LIN {X -5606.996,Y 2667.355,Z 190.712,A 89.99946,B 0.00000,C 180.00000} ; preinsert
  LIN {X -5606.996,Y 2667.355,Z -59.288,A 89.99946,B 0.00000,C 180.00000} ; insert
  LIN {X -5606.996,Y 2667.355,Z -59.288,A 89.99946,B 0.00000,C 180.00000} ; release
  LIN {X -5606.996,Y 2667.355,Z 240.712,A 89.99946,B 0.00000,C 180.00000} ; retreat
  ; Step 2310, bar 703
  LIN {X -5481.996,Y 2667.355,Z 1143.930,A 89.99946,B 0.00000,C 180.00000} ; outside
  LIN {X -5481.996,Y 2667.355,Z 190.712,A 89.99946,B 0.00000,C 180.00000} ; preinsert
  LIN {X -5481.996,Y 2667.355,Z -59.288,A 89.99946,B 0.00000,C 180.00000} ; insert
  LIN {X -5481.996,Y 2667.355,Z -59.288,A 89.99946,B 0.00000,C 180.00000} ; release
  LIN {X -5481.996,Y 2667.355,Z 240.712,A 89.99946,B 0.00000,C 180.00000} ; retreat
  ; Step 2311, bar 701
  LIN {X -5356.996,Y 2667.355,Z 1143.930,A 89.99946,B 0.00000,C 180.00000} ; outside
  LIN {X -5356.996,Y 2667.355,Z 190.712,A 89.99946,B 0.00000,C 180.00000} ; preinsert
  LIN {X -5356.996,Y 2667.355,Z -59.288,A 89.99946,B 0.00000,C 180.00000} ; insert
  LIN {X -5356.996,Y 2667.355,Z -59.288,A 89.99946,B 0.00000,C 180.00000} ; release
  LIN {X -5356.996,Y 2667.355,Z 240.712,A 89.99946,B 0.00000,C 180.00000} ; retreat
  ; Step 2312, bar 699
  LIN {X -5231.996,Y 2667.355,Z 1143.930,A 89.99946,B 0.00000,C 180.00000} ; outside
  LIN {X -5231.996,Y 2667.355,Z 190.712,A 89.99946,B 0.00000,C 180.00000} ; preinsert
  LIN {X -5231.996,Y 2667.355,Z -59.288,A 89.99946,B 0.00000,C 180.00000} ; insert
  LIN {X -5231.996,Y 2667.355,Z -59.288,A 89.99946,B 0.00000,C 180.00000} ; release
  LIN {X -5231.996,Y 2667.355,Z 240.712,A 89.99946,B 0.00000,C 180.00000} ; retreat
  ; Step 2313, bar 697
  LIN {X -5106.996,Y 2667.355,Z 1143.930,A 89.99946,B 0.00000,C 180.00000} ; outside
  LIN {X -5106.996,Y 2667.355,Z 190.712,A 89.99946,B 0.00000,C 180.00000} ; preinsert
  LIN {X -5106.996,Y 2667.355,Z -59.288,A 89.99946,B 0.00000,C 180.00000} ; insert
  LIN {X -5106.996,Y 2667.355,Z -59.288,A 89.99946,B 0.00000,C 180.00000} ; release
  LIN {X -5106.996,Y 2667.355,Z 240.712,A 89.99946,B 0.00000,C 180.00000} ; retreat
  ; Step 2314, bar 695
  LIN {X -4981.996,Y 2667.355,Z 1143.930,A 89.99946,B 0.00000,C 180.00000} ; outside
  LIN {X -4981.996,Y 2667.355,Z 190.712,A 89.99946,B 0.00000,C 180.00000} ; preinsert
  LIN {X -4981.996,Y 2667.355,Z -59.288,A 89.99946,B 0.00000,C 180.00000} ; insert
  LIN {X -4981.996,Y 2667.355,Z -59.288,A 89.99946,B 0.00000,C 180.00000} ; release
  LIN {X -4981.996,Y 2667.355,Z 240.712,A 89.99946,B 0.00000,C 180.00000} ; retreat
  ; Step 2315, bar 693
  LIN {X -4856.996,Y 2667.355,Z 1143.930,A 89.99946,B 0.00000,C 180.00000} ; outside
  LIN {X -4856.996,Y 2667.355,Z 190.712,A 89.99946,B 0.00000,C 180.00000} ; preinsert
  LIN {X -4856.996,Y 2667.355,Z -59.288,A 89.99946,B 0.00000,C 180.00000} ; insert
  LIN {X -4856.996,Y 2667.355,Z -59.288,A 89.99946,B 0.00000,C 180.00000} ; release
  LIN {X -4856.996,Y 2667.355,Z 240.712,A 89.99946,B 0.00000,C 180.00000} ; retreat
  ; Step 2316, bar 691
  LIN {X -4731.996,Y 2667.355,Z 1143.930,A 89.99946,B 0.00000,C 180.00000} ; outside
  LIN {X -4731.996,Y 2667.355,Z 190.712,A 89.99946,B 0.00000,C 180.00000} ; preinsert
  LIN {X -4731.996,Y 2667.355,Z -59.288,A 89.99946,B 0.00000,C 180.00000} ; insert
  LIN {X -4731.996,Y 2667.355,Z -59.288,A 89.99946,B 0.00000,C 180.00000} ; release
  LIN {X -4731.996,Y 2667.355,Z 240.712,A 89.99946,B 0.00000,C 180.00000} ; retreat
  ; Step 2317, bar 689
  LIN {X -4606.996,Y 2667.355,Z 1143.930,A 89.99946,B 0.00000,C 180.00000} ; outside
  LIN {X -4606.996,Y 2667.355,Z 190.712,A 89.99946,B 0.00000,C 180.00000} ; preinsert
  LIN {X -4606.996,Y 2667.355,Z -59.288,A 89.99946,B 0.00000,C 180.00000} ; insert
  LIN {X -4606.996,Y 2667.355,Z -59.288,A 89.99946,B 0.00000,C 180.00000} ; release
  LIN {X -4606.996,Y 2667.355,Z 240.712,A 89.99946,B 0.00000,C 180.00000} ; retreat
  ; Step 2318, bar 687
  LIN {X -4481.996,Y 2667.355,Z 1143.930,A 89.99946,B 0.00000,C 180.00000} ; outside
  LIN {X -4481.996,Y 2667.355,Z 190.712,A 89.99946,B 0.00000,C 180.00000} ; preinsert
  LIN {X -4481.996,Y 2667.355,Z -59.288,A 89.99946,B 0.00000,C 180.00000} ; insert
  LIN {X -4481.996,Y 2667.355,Z -59.288,A 89.99946,B 0.00000,C 180.00000} ; release
  LIN {X -4481.996,Y 2667.355,Z 240.712,A 89.99946,B 0.00000,C 180.00000} ; retreat
  ; Step 2319, bar 685
  LIN {X -4356.996,Y 2667.355,Z 1143.930,A 89.99946,B 0.00000,C 180.00000} ; outside
  LIN {X -4356.996,Y 2667.355,Z 190.712,A 89.99946,B 0.00000,C 180.00000} ; preinsert
  LIN {X -4356.996,Y 2667.355,Z -59.288,A 89.99946,B 0.00000,C 180.00000} ; insert
  LIN {X -4356.996,Y 2667.355,Z -59.288,A 89.99946,B 0.00000,C 180.00000} ; release
  LIN {X -4356.996,Y 2667.355,Z 240.712,A 89.99946,B 0.00000,C 180.00000} ; retreat
  ; Step 2320, bar 683
  LIN {X -4231.996,Y 2667.355,Z 1143.930,A 89.99946,B 0.00000,C 180.00000} ; outside
  LIN {X -4231.996,Y 2667.355,Z 190.712,A 89.99946,B 0.00000,C 180.00000} ; preinsert
  LIN {X -4231.996,Y 2667.355,Z -59.288,A 89.99946,B 0.00000,C 180.00000} ; insert
  LIN {X -4231.996,Y 2667.355,Z -59.288,A 89.99946,B 0.00000,C 180.00000} ; release
  LIN {X -4231.996,Y 2667.355,Z 240.712,A 89.99946,B 0.00000,C 180.00000} ; retreat
  ; Step 2321, bar 681
  LIN {X -4106.996,Y 2667.355,Z 1143.930,A 89.99946,B 0.00000,C 180.00000} ; outside
  LIN {X -4106.996,Y 2667.355,Z 190.712,A 89.99946,B 0.00000,C 180.00000} ; preinsert
  LIN {X -4106.996,Y 2667.355,Z -59.288,A 89.99946,B 0.00000,C 180.00000} ; insert
  LIN {X -4106.996,Y 2667.355,Z -59.288,A 89.99946,B 0.00000,C 180.00000} ; release
  LIN {X -4106.996,Y 2667.355,Z 240.712,A 89.99946,B 0.00000,C 180.00000} ; retreat
  ; Step 2322, bar 679
  LIN {X -3981.996,Y 2667.355,Z 1143.930,A 89.99946,B 0.00000,C 180.00000} ; outside
  LIN {X -3981.996,Y 2667.355,Z 190.712,A 89.99946,B 0.00000,C 180.00000} ; preinsert
  LIN {X -3981.996,Y 2667.355,Z -59.288,A 89.99946,B 0.00000,C 180.00000} ; insert
  LIN {X -3981.996,Y 2667.355,Z -59.288,A 89.99946,B 0.00000,C 180.00000} ; release
  LIN {X -3981.996,Y 2667.355,Z 240.712,A 89.99946,B 0.00000,C 180.00000} ; retreat
  ; Step 2323, bar 677
  LIN {X -3856.996,Y 2667.355,Z 1143.930,A 89.99946,B 0.00000,C 180.00000} ; outside
  LIN {X -3856.996,Y 2667.355,Z 190.712,A 89.99946,B 0.00000,C 180.00000} ; preinsert
  LIN {X -3856.996,Y 2667.355,Z -59.288,A 89.99946,B 0.00000,C 180.00000} ; insert
  LIN {X -3856.996,Y 2667.355,Z -59.288,A 89.99946,B 0.00000,C 180.00000} ; release
  LIN {X -3856.996,Y 2667.355,Z 240.712,A 89.99946,B 0.00000,C 180.00000} ; retreat
  ; Step 2324, bar 675
  LIN {X -3731.996,Y 2667.355,Z 1143.930,A 89.99946,B 0.00000,C 180.00000} ; outside
  LIN {X -3731.996,Y 2667.355,Z 190.712,A 89.99946,B 0.00000,C 180.00000} ; preinsert
  LIN {X -3731.996,Y 2667.355,Z -59.288,A 89.99946,B 0.00000,C 180.00000} ; insert
  LIN {X -3731.996,Y 2667.355,Z -59.288,A 89.99946,B 0.00000,C 180.00000} ; release
  LIN {X -3731.996,Y 2667.355,Z 240.712,A 89.99946,B 0.00000,C 180.00000} ; retreat
  ; Step 2325, bar 673
  LIN {X -3606.996,Y 2667.355,Z 1143.930,A 89.99946,B 0.00000,C 180.00000} ; outside
  LIN {X -3606.996,Y 2667.355,Z 190.712,A 89.99946,B 0.00000,C 180.00000} ; preinsert
  LIN {X -3606.996,Y 2667.355,Z -59.288,A 89.99946,B 0.00000,C 180.00000} ; insert
  LIN {X -3606.996,Y 2667.355,Z -59.288,A 89.99946,B 0.00000,C 180.00000} ; release
  LIN {X -3606.996,Y 2667.355,Z 240.712,A 89.99946,B 0.00000,C 180.00000} ; retreat
  ; Step 2326, bar 671
  LIN {X -3481.996,Y 2667.355,Z 1143.930,A 89.99946,B 0.00000,C 180.00000} ; outside
  LIN {X -3481.996,Y 2667.355,Z 190.712,A 89.99946,B 0.00000,C 180.00000} ; preinsert
  LIN {X -3481.996,Y 2667.355,Z -59.288,A 89.99946,B 0.00000,C 180.00000} ; insert
  LIN {X -3481.996,Y 2667.355,Z -59.288,A 89.99946,B 0.00000,C 180.00000} ; release
  LIN {X -3481.996,Y 2667.355,Z 240.712,A 89.99946,B 0.00000,C 180.00000} ; retreat
  ; Step 2327, bar 669
  LIN {X -3356.996,Y 2667.355,Z 1143.930,A 89.99946,B 0.00000,C 180.00000} ; outside
  LIN {X -3356.996,Y 2667.355,Z 190.712,A 89.99946,B 0.00000,C 180.00000} ; preinsert
  LIN {X -3356.996,Y 2667.355,Z -59.288,A 89.99946,B 0.00000,C 180.00000} ; insert
  LIN {X -3356.996,Y 2667.355,Z -59.288,A 89.99946,B 0.00000,C 180.00000} ; release
  LIN {X -3356.996,Y 2667.355,Z 240.712,A 89.99946,B 0.00000,C 180.00000} ; retreat
  ; Step 2328, bar 667
  LIN {X -3231.996,Y 2667.355,Z 1143.930,A 89.99946,B 0.00000,C 180.00000} ; outside
  LIN {X -3231.996,Y 2667.355,Z 190.712,A 89.99946,B 0.00000,C 180.00000} ; preinsert
  LIN {X -3231.996,Y 2667.355,Z -59.288,A 89.99946,B 0.00000,C 180.00000} ; insert
  LIN {X -3231.996,Y 2667.355,Z -59.288,A 89.99946,B 0.00000,C 180.00000} ; release
  LIN {X -3231.996,Y 2667.355,Z 240.712,A 89.99946,B 0.00000,C 180.00000} ; retreat
  ; Step 2329, bar 665
  LIN {X -3106.996,Y 2667.355,Z 1143.930,A 89.99946,B 0.00000,C 180.00000} ; outside
  LIN {X -3106.996,Y 2667.355,Z 190.712,A 89.99946,B 0.00000,C 180.00000} ; preinsert
  LIN {X -3106.996,Y 2667.355,Z -59.288,A 89.99946,B 0.00000,C 180.00000} ; insert
  LIN {X -3106.996,Y 2667.355,Z -59.288,A 89.99946,B 0.00000,C 180.00000} ; release
  LIN {X -3106.996,Y 2667.355,Z 240.712,A 89.99946,B 0.00000,C 180.00000} ; retreat
  ; Step 2330, bar 663
  LIN {X -2981.996,Y 2667.355,Z 1143.930,A 89.99946,B 0.00000,C 180.00000} ; outside
  LIN {X -2981.996,Y 2667.355,Z 190.712,A 89.99946,B 0.00000,C 180.00000} ; preinsert
  LIN {X -2981.996,Y 2667.355,Z -59.288,A 89.99946,B 0.00000,C 180.00000} ; insert
  LIN {X -2981.996,Y 2667.355,Z -59.288,A 89.99946,B 0.00000,C 180.00000} ; release
  LIN {X -2981.996,Y 2667.355,Z 240.712,A 89.99946,B 0.00000,C 180.00000} ; retreat
  ; Step 2331, bar 661
  LIN {X -2856.996,Y 2667.355,Z 1143.930,A 89.99946,B 0.00000,C 180.00000} ; outside
  LIN {X -2856.996,Y 2667.355,Z 190.712,A 89.99946,B 0.00000,C 180.00000} ; preinsert
  LIN {X -2856.996,Y 2667.355,Z -59.288,A 89.99946,B 0.00000,C 180.00000} ; insert
  LIN {X -2856.996,Y 2667.355,Z -59.288,A 89.99946,B 0.00000,C 180.00000} ; release
  LIN {X -2856.996,Y 2667.355,Z 240.712,A 89.99946,B 0.00000,C 180.00000} ; retreat
  ; Step 2332, bar 659
  LIN {X -2731.996,Y 2667.355,Z 1143.930,A 89.99946,B 0.00000,C 180.00000} ; outside
  LIN {X -2731.996,Y 2667.355,Z 190.712,A 89.99946,B 0.00000,C 180.00000} ; preinsert
  LIN {X -2731.996,Y 2667.355,Z -59.288,A 89.99946,B 0.00000,C 180.00000} ; insert
  LIN {X -2731.996,Y 2667.355,Z -59.288,A 89.99946,B 0.00000,C 180.00000} ; release
  LIN {X -2731.996,Y 2667.355,Z 240.712,A 89.99946,B 0.00000,C 180.00000} ; retreat
  ; Step 2333, bar 657
  LIN {X -2606.996,Y 2667.355,Z 1143.930,A 89.99946,B 0.00000,C 180.00000} ; outside
  LIN {X -2606.996,Y 2667.355,Z 190.712,A 89.99946,B 0.00000,C 180.00000} ; preinsert
  LIN {X -2606.996,Y 2667.355,Z -59.288,A 89.99946,B 0.00000,C 180.00000} ; insert
  LIN {X -2606.996,Y 2667.355,Z -59.288,A 89.99946,B 0.00000,C 180.00000} ; release
  LIN {X -2606.996,Y 2667.355,Z 240.712,A 89.99946,B 0.00000,C 180.00000} ; retreat
  ; Step 2334, bar 655
  LIN {X -2481.996,Y 2667.355,Z 1143.930,A 89.99946,B 0.00000,C 180.00000} ; outside
  LIN {X -2481.996,Y 2667.355,Z 190.712,A 89.99946,B 0.00000,C 180.00000} ; preinsert
  LIN {X -2481.996,Y 2667.355,Z -59.288,A 89.99946,B 0.00000,C 180.00000} ; insert
  LIN {X -2481.996,Y 2667.355,Z -59.288,A 89.99946,B 0.00000,C 180.00000} ; release
  LIN {X -2481.996,Y 2667.355,Z 240.712,A 89.99946,B 0.00000,C 180.00000} ; retreat
  ; Step 2335, bar 653
  LIN {X -2356.996,Y 2667.355,Z 1143.930,A 89.99946,B 0.00000,C 180.00000} ; outside
  LIN {X -2356.996,Y 2667.355,Z 190.712,A 89.99946,B 0.00000,C 180.00000} ; preinsert
  LIN {X -2356.996,Y 2667.355,Z -59.288,A 89.99946,B 0.00000,C 180.00000} ; insert
  LIN {X -2356.996,Y 2667.355,Z -59.288,A 89.99946,B 0.00000,C 180.00000} ; release
  LIN {X -2356.996,Y 2667.355,Z 240.712,A 89.99946,B 0.00000,C 180.00000} ; retreat
  ; Step 2336, bar 651
  LIN {X -2231.996,Y 2667.355,Z 1143.930,A 89.99946,B 0.00000,C 180.00000} ; outside
  LIN {X -2231.996,Y 2667.355,Z 190.712,A 89.99946,B 0.00000,C 180.00000} ; preinsert
  LIN {X -2231.996,Y 2667.355,Z -59.288,A 89.99946,B 0.00000,C 180.00000} ; insert
  LIN {X -2231.996,Y 2667.355,Z -59.288,A 89.99946,B 0.00000,C 180.00000} ; release
  LIN {X -2231.996,Y 2667.355,Z 240.712,A 89.99946,B 0.00000,C 180.00000} ; retreat
  ; Step 2337, bar 649
  LIN {X -2106.996,Y 2667.355,Z 1143.930,A 89.99946,B 0.00000,C 180.00000} ; outside
  LIN {X -2106.996,Y 2667.355,Z 190.712,A 89.99946,B 0.00000,C 180.00000} ; preinsert
  LIN {X -2106.996,Y 2667.355,Z -59.288,A 89.99946,B 0.00000,C 180.00000} ; insert
  LIN {X -2106.996,Y 2667.355,Z -59.288,A 89.99946,B 0.00000,C 180.00000} ; release
  LIN {X -2106.996,Y 2667.355,Z 240.712,A 89.99946,B 0.00000,C 180.00000} ; retreat
  ; Step 2338, bar 647
  LIN {X -1856.996,Y 2667.355,Z 1143.930,A 89.99946,B 0.00000,C 180.00000} ; outside
  LIN {X -1856.996,Y 2667.355,Z 190.712,A 89.99946,B 0.00000,C 180.00000} ; preinsert
  LIN {X -1856.996,Y 2667.355,Z -59.288,A 89.99946,B 0.00000,C 180.00000} ; insert
  LIN {X -1856.996,Y 2667.355,Z -59.288,A 89.99946,B 0.00000,C 180.00000} ; release
  LIN {X -1856.996,Y 2667.355,Z 240.712,A 89.99946,B 0.00000,C 180.00000} ; retreat
  ; Step 2339, bar 645
  LIN {X -1731.996,Y 2667.355,Z 1143.930,A 89.99946,B 0.00000,C 180.00000} ; outside
  LIN {X -1731.996,Y 2667.355,Z 190.712,A 89.99946,B 0.00000,C 180.00000} ; preinsert
  LIN {X -1731.996,Y 2667.355,Z -59.288,A 89.99946,B 0.00000,C 180.00000} ; insert
  LIN {X -1731.996,Y 2667.355,Z -59.288,A 89.99946,B 0.00000,C 180.00000} ; release
  LIN {X -1731.996,Y 2667.355,Z 240.712,A 89.99946,B 0.00000,C 180.00000} ; retreat
  ; Step 2340, bar 643
  LIN {X -1606.996,Y 2667.355,Z 1143.930,A 89.99946,B 0.00000,C 180.00000} ; outside
  LIN {X -1606.996,Y 2667.355,Z 190.712,A 89.99946,B 0.00000,C 180.00000} ; preinsert
  LIN {X -1606.996,Y 2667.355,Z -59.288,A 89.99946,B 0.00000,C 180.00000} ; insert
  LIN {X -1606.996,Y 2667.355,Z -59.288,A 89.99946,B 0.00000,C 180.00000} ; release
  LIN {X -1606.996,Y 2667.355,Z 240.712,A 89.99946,B 0.00000,C 180.00000} ; retreat
  ; Step 2341, bar 641
  LIN {X -1481.996,Y 2667.355,Z 1143.930,A 89.99946,B 0.00000,C 180.00000} ; outside
  LIN {X -1481.996,Y 2667.355,Z 190.712,A 89.99946,B 0.00000,C 180.00000} ; preinsert
  LIN {X -1481.996,Y 2667.355,Z -59.288,A 89.99946,B 0.00000,C 180.00000} ; insert
  LIN {X -1481.996,Y 2667.355,Z -59.288,A 89.99946,B 0.00000,C 180.00000} ; release
  LIN {X -1481.996,Y 2667.355,Z 240.712,A 89.99946,B 0.00000,C 180.00000} ; retreat
  ; Step 2342, bar 639
  LIN {X -1356.996,Y 2667.355,Z 1143.930,A 89.99946,B 0.00000,C 180.00000} ; outside
  LIN {X -1356.996,Y 2667.355,Z 190.712,A 89.99946,B 0.00000,C 180.00000} ; preinsert
  LIN {X -1356.996,Y 2667.355,Z -59.288,A 89.99946,B 0.00000,C 180.00000} ; insert
  LIN {X -1356.996,Y 2667.355,Z -59.288,A 89.99946,B 0.00000,C 180.00000} ; release
  LIN {X -1356.996,Y 2667.355,Z 240.712,A 89.99946,B 0.00000,C 180.00000} ; retreat
  ; Step 2343, bar 637
  LIN {X -1231.996,Y 2667.355,Z 1143.930,A 89.99946,B 0.00000,C 180.00000} ; outside
  LIN {X -1231.996,Y 2667.355,Z 190.712,A 89.99946,B 0.00000,C 180.00000} ; preinsert
  LIN {X -1231.996,Y 2667.355,Z -59.288,A 89.99946,B 0.00000,C 180.00000} ; insert
  LIN {X -1231.996,Y 2667.355,Z -59.288,A 89.99946,B 0.00000,C 180.00000} ; release
  LIN {X -1231.996,Y 2667.355,Z 240.712,A 89.99946,B 0.00000,C 180.00000} ; retreat
  ; Step 2344, bar 635
  LIN {X -1106.996,Y 2667.355,Z 1143.930,A 89.99946,B 0.00000,C 180.00000} ; outside
  LIN {X -1106.996,Y 2667.355,Z 190.712,A 89.99946,B 0.00000,C 180.00000} ; preinsert
  LIN {X -1106.996,Y 2667.355,Z -59.288,A 89.99946,B 0.00000,C 180.00000} ; insert
  LIN {X -1106.996,Y 2667.355,Z -59.288,A 89.99946,B 0.00000,C 180.00000} ; release
  LIN {X -1106.996,Y 2667.355,Z 240.712,A 89.99946,B 0.00000,C 180.00000} ; retreat
  ; Step 2345, bar 633
  LIN {X -981.996,Y 2667.355,Z 1143.930,A 89.99946,B 0.00000,C 180.00000} ; outside
  LIN {X -981.996,Y 2667.355,Z 190.712,A 89.99946,B 0.00000,C 180.00000} ; preinsert
  LIN {X -981.996,Y 2667.355,Z -59.288,A 89.99946,B 0.00000,C 180.00000} ; insert
  LIN {X -981.996,Y 2667.355,Z -59.288,A 89.99946,B 0.00000,C 180.00000} ; release
  LIN {X -981.996,Y 2667.355,Z 240.712,A 89.99946,B 0.00000,C 180.00000} ; retreat
  ; Step 2346, bar 631
  LIN {X -856.996,Y 2667.355,Z 1143.930,A 89.99946,B 0.00000,C 180.00000} ; outside
  LIN {X -856.996,Y 2667.355,Z 190.712,A 89.99946,B 0.00000,C 180.00000} ; preinsert
  LIN {X -856.996,Y 2667.355,Z -59.288,A 89.99946,B 0.00000,C 180.00000} ; insert
  LIN {X -856.996,Y 2667.355,Z -59.288,A 89.99946,B 0.00000,C 180.00000} ; release
  LIN {X -856.996,Y 2667.355,Z 240.712,A 89.99946,B 0.00000,C 180.00000} ; retreat
  ; Step 2347, bar 629
  LIN {X -731.996,Y 2667.355,Z 1143.930,A 89.99946,B 0.00000,C 180.00000} ; outside
  LIN {X -731.996,Y 2667.355,Z 190.712,A 89.99946,B 0.00000,C 180.00000} ; preinsert
  LIN {X -731.996,Y 2667.355,Z -59.288,A 89.99946,B 0.00000,C 180.00000} ; insert
  LIN {X -731.996,Y 2667.355,Z -59.288,A 89.99946,B 0.00000,C 180.00000} ; release
  LIN {X -731.996,Y 2667.355,Z 240.712,A 89.99946,B 0.00000,C 180.00000} ; retreat
  ; Step 2348, bar 627
  LIN {X -606.996,Y 2667.355,Z 1143.930,A 89.99946,B 0.00000,C 180.00000} ; outside
  LIN {X -606.996,Y 2667.355,Z 190.712,A 89.99946,B 0.00000,C 180.00000} ; preinsert
  LIN {X -606.996,Y 2667.355,Z -59.288,A 89.99946,B 0.00000,C 180.00000} ; insert
  LIN {X -606.996,Y 2667.355,Z -59.288,A 89.99946,B 0.00000,C 180.00000} ; release
  LIN {X -606.996,Y 2667.355,Z 240.712,A 89.99946,B 0.00000,C 180.00000} ; retreat
  ; Step 2349, bar 625
  LIN {X -481.996,Y 2667.355,Z 1143.930,A 89.99946,B 0.00000,C 180.00000} ; outside
  LIN {X -481.996,Y 2667.355,Z 190.712,A 89.99946,B 0.00000,C 180.00000} ; preinsert
  LIN {X -481.996,Y 2667.355,Z -59.288,A 89.99946,B 0.00000,C 180.00000} ; insert
  LIN {X -481.996,Y 2667.355,Z -59.288,A 89.99946,B 0.00000,C 180.00000} ; release
  LIN {X -481.996,Y 2667.355,Z 240.712,A 89.99946,B 0.00000,C 180.00000} ; retreat
  ; Step 2350, bar 623
  LIN {X -356.996,Y 2667.355,Z 1143.930,A 89.99946,B 0.00000,C 180.00000} ; outside
  LIN {X -356.996,Y 2667.355,Z 190.712,A 89.99946,B 0.00000,C 180.00000} ; preinsert
  LIN {X -356.996,Y 2667.355,Z -59.288,A 89.99946,B 0.00000,C 180.00000} ; insert
  LIN {X -356.996,Y 2667.355,Z -59.288,A 89.99946,B 0.00000,C 180.00000} ; release
  LIN {X -356.996,Y 2667.355,Z 240.712,A 89.99946,B 0.00000,C 180.00000} ; retreat
  ; Step 2351, bar 621
  LIN {X -231.996,Y 2667.355,Z 1143.930,A 89.99946,B 0.00000,C 180.00000} ; outside
  LIN {X -231.996,Y 2667.355,Z 190.712,A 89.99946,B 0.00000,C 180.00000} ; preinsert
  LIN {X -231.996,Y 2667.355,Z -59.288,A 89.99946,B 0.00000,C 180.00000} ; insert
  LIN {X -231.996,Y 2667.355,Z -59.288,A 89.99946,B 0.00000,C 180.00000} ; release
  LIN {X -231.996,Y 2667.355,Z 240.712,A 89.99946,B 0.00000,C 180.00000} ; retreat
  ; Step 2352, bar 619
  LIN {X -106.996,Y 2667.355,Z 1143.930,A 89.99946,B 0.00000,C 180.00000} ; outside
  LIN {X -106.996,Y 2667.355,Z 190.712,A 89.99946,B 0.00000,C 180.00000} ; preinsert
  LIN {X -106.996,Y 2667.355,Z -59.288,A 89.99946,B 0.00000,C 180.00000} ; insert
  LIN {X -106.996,Y 2667.355,Z -59.288,A 89.99946,B 0.00000,C 180.00000} ; release
  LIN {X -106.996,Y 2667.355,Z 240.712,A 89.99946,B 0.00000,C 180.00000} ; retreat
  ; Step 2353, bar 610
  LIN {X -14031.817,Y -2845.819,Z 1147.317,A 90.02227,B 0.00000,C 180.00000} ; outside
  LIN {X -14031.817,Y -2845.819,Z 194.063,A 90.02227,B 0.00000,C 180.00000} ; preinsert
  LIN {X -14031.817,Y -2845.819,Z -55.937,A 90.02227,B 0.00000,C 180.00000} ; insert
  LIN {X -14031.817,Y -2845.819,Z -55.937,A 90.02227,B 0.00000,C 180.00000} ; release
  LIN {X -14031.817,Y -2845.819,Z 244.063,A 90.02227,B 0.00000,C 180.00000} ; retreat
  ; Step 2354, bar 608
  LIN {X -13931.817,Y -2845.819,Z 1147.317,A 90.02227,B 0.00000,C 180.00000} ; outside
  LIN {X -13931.817,Y -2845.819,Z 194.063,A 90.02227,B 0.00000,C 180.00000} ; preinsert
  LIN {X -13931.817,Y -2845.819,Z -55.937,A 90.02227,B 0.00000,C 180.00000} ; insert
  LIN {X -13931.817,Y -2845.819,Z -55.937,A 90.02227,B 0.00000,C 180.00000} ; release
  LIN {X -13931.817,Y -2845.819,Z 244.063,A 90.02227,B 0.00000,C 180.00000} ; retreat
  ; Step 2355, bar 614
  LIN {X -9981.817,Y -2845.819,Z 1147.317,A 90.02227,B 0.00000,C 180.00000} ; outside
  LIN {X -9981.817,Y -2845.819,Z 194.063,A 90.02227,B 0.00000,C 180.00000} ; preinsert
  LIN {X -9981.817,Y -2845.819,Z -55.937,A 90.02227,B 0.00000,C 180.00000} ; insert
  LIN {X -9981.817,Y -2845.819,Z -55.937,A 90.02227,B 0.00000,C 180.00000} ; release
  LIN {X -9981.817,Y -2845.819,Z 244.063,A 90.02227,B 0.00000,C 180.00000} ; retreat
  ; Step 2356, bar 612
  LIN {X -5981.817,Y -2845.819,Z 1147.317,A 90.02227,B 0.00000,C 180.00000} ; outside
  LIN {X -5981.817,Y -2845.819,Z 194.063,A 90.02227,B 0.00000,C 180.00000} ; preinsert
  LIN {X -5981.817,Y -2845.819,Z -55.937,A 90.02227,B 0.00000,C 180.00000} ; insert
  LIN {X -5981.817,Y -2845.819,Z -55.937,A 90.02227,B 0.00000,C 180.00000} ; release
  LIN {X -5981.817,Y -2845.819,Z 244.063,A 90.02227,B 0.00000,C 180.00000} ; retreat
  ; Step 2357, bar 616
  LIN {X -1981.817,Y -2845.819,Z 1147.317,A 90.02227,B 0.00000,C 180.00000} ; outside
  LIN {X -1981.817,Y -2845.819,Z 194.063,A 90.02227,B 0.00000,C 180.00000} ; preinsert
  LIN {X -1981.817,Y -2845.819,Z -55.937,A 90.02227,B 0.00000,C 180.00000} ; insert
  LIN {X -1981.817,Y -2845.819,Z -55.937,A 90.02227,B 0.00000,C 180.00000} ; release
  LIN {X -1981.817,Y -2845.819,Z 244.063,A 90.02227,B 0.00000,C 180.00000} ; retreat
  ; Step 2358, bar 607
  LIN {X 1981.817,Y 2845.819,Z 1147.317,A -89.97773,B 0.00000,C 180.00000} ; outside
  LIN {X 1981.817,Y 2845.819,Z 194.063,A -89.97773,B 0.00000,C 180.00000} ; preinsert
  LIN {X 1981.817,Y 2845.819,Z -55.937,A -89.97773,B 0.00000,C 180.00000} ; insert
  LIN {X 1981.817,Y 2845.819,Z -55.937,A -89.97773,B 0.00000,C 180.00000} ; release
  LIN {X 1981.817,Y 2845.819,Z 244.063,A -89.97773,B 0.00000,C 180.00000} ; retreat
  ; Step 2359, bar 603
  LIN {X 5981.817,Y 2845.819,Z 1147.317,A -89.97773,B 0.00000,C 180.00000} ; outside
  LIN {X 5981.817,Y 2845.819,Z 194.063,A -89.97773,B 0.00000,C 180.00000} ; preinsert
  LIN {X 5981.817,Y 2845.819,Z -55.937,A -89.97773,B 0.00000,C 180.00000} ; insert
  LIN {X 5981.817,Y 2845.819,Z -55.937,A -89.97773,B 0.00000,C 180.00000} ; release
  LIN {X 5981.817,Y 2845.819,Z 244.063,A -89.97773,B 0.00000,C 180.00000} ; retreat
  ; Step 2360, bar 605
  LIN {X 9981.817,Y 2845.819,Z 1147.317,A -89.97773,B 0.00000,C 180.00000} ; outside
  LIN {X 9981.817,Y 2845.819,Z 194.063,A -89.97773,B 0.00000,C 180.00000} ; preinsert
  LIN {X 9981.817,Y 2845.819,Z -55.937,A -89.97773,B 0.00000,C 180.00000} ; insert
  LIN {X 9981.817,Y 2845.819,Z -55.937,A -89.97773,B 0.00000,C 180.00000} ; release
  LIN {X 9981.817,Y 2845.819,Z 244.063,A -89.97773,B 0.00000,C 180.00000} ; retreat
  ; Step 2361, bar 599
  LIN {X 13931.817,Y 2845.819,Z 1147.317,A -89.97773,B 0.00000,C 180.00000} ; outside
  LIN {X 13931.817,Y 2845.819,Z 194.063,A -89.97773,B 0.00000,C 180.00000} ; preinsert
  LIN {X 13931.817,Y 2845.819,Z -55.937,A -89.97773,B 0.00000,C 180.00000} ; insert
  LIN {X 13931.817,Y 2845.819,Z -55.937,A -89.97773,B 0.00000,C 180.00000} ; release
  LIN {X 13931.817,Y 2845.819,Z 244.063,A -89.97773,B 0.00000,C 180.00000} ; retreat
  ; Step 2362, bar 601
  LIN {X 14031.817,Y 2845.819,Z 1147.317,A -89.97773,B 0.00000,C 180.00000} ; outside
  LIN {X 14031.817,Y 2845.819,Z 194.063,A -89.97773,B 0.00000,C 180.00000} ; preinsert
  LIN {X 14031.817,Y 2845.819,Z -55.937,A -89.97773,B 0.00000,C 180.00000} ; insert
  LIN {X 14031.817,Y 2845.819,Z -55.937,A -89.97773,B 0.00000,C 180.00000} ; release
  LIN {X 14031.817,Y 2845.819,Z 244.063,A -89.97773,B 0.00000,C 180.00000} ; retreat
  ; Step 2363, bar 606
  LIN {X 1981.817,Y -2845.819,Z 1147.317,A 89.97773,B 0.00000,C 180.00000} ; outside
  LIN {X 1981.817,Y -2845.819,Z 194.063,A 89.97773,B 0.00000,C 180.00000} ; preinsert
  LIN {X 1981.817,Y -2845.819,Z -55.937,A 89.97773,B 0.00000,C 180.00000} ; insert
  LIN {X 1981.817,Y -2845.819,Z -55.937,A 89.97773,B 0.00000,C 180.00000} ; release
  LIN {X 1981.817,Y -2845.819,Z 244.063,A 89.97773,B 0.00000,C 180.00000} ; retreat
  ; Step 2364, bar 602
  LIN {X 5981.817,Y -2845.819,Z 1147.317,A 89.97773,B 0.00000,C 180.00000} ; outside
  LIN {X 5981.817,Y -2845.819,Z 194.063,A 89.97773,B 0.00000,C 180.00000} ; preinsert
  LIN {X 5981.817,Y -2845.819,Z -55.937,A 89.97773,B 0.00000,C 180.00000} ; insert
  LIN {X 5981.817,Y -2845.819,Z -55.937,A 89.97773,B 0.00000,C 180.00000} ; release
  LIN {X 5981.817,Y -2845.819,Z 244.063,A 89.97773,B 0.00000,C 180.00000} ; retreat
  ; Step 2365, bar 604
  LIN {X 9981.817,Y -2845.819,Z 1147.317,A 89.97773,B 0.00000,C 180.00000} ; outside
  LIN {X 9981.817,Y -2845.819,Z 194.063,A 89.97773,B 0.00000,C 180.00000} ; preinsert
  LIN {X 9981.817,Y -2845.819,Z -55.937,A 89.97773,B 0.00000,C 180.00000} ; insert
  LIN {X 9981.817,Y -2845.819,Z -55.937,A 89.97773,B 0.00000,C 180.00000} ; release
  LIN {X 9981.817,Y -2845.819,Z 244.063,A 89.97773,B 0.00000,C 180.00000} ; retreat
  ; Step 2366, bar 598
  LIN {X 13931.817,Y -2845.819,Z 1147.317,A 89.97773,B 0.00000,C 180.00000} ; outside
  LIN {X 13931.817,Y -2845.819,Z 194.063,A 89.97773,B 0.00000,C 180.00000} ; preinsert
  LIN {X 13931.817,Y -2845.819,Z -55.937,A 89.97773,B 0.00000,C 180.00000} ; insert
  LIN {X 13931.817,Y -2845.819,Z -55.937,A 89.97773,B 0.00000,C 180.00000} ; release
  LIN {X 13931.817,Y -2845.819,Z 244.063,A 89.97773,B 0.00000,C 180.00000} ; retreat
  ; Step 2367, bar 600
  LIN {X 14031.817,Y -2845.819,Z 1147.317,A 89.97773,B 0.00000,C 180.00000} ; outside
  LIN {X 14031.817,Y -2845.819,Z 194.063,A 89.97773,B 0.00000,C 180.00000} ; preinsert
  LIN {X 14031.817,Y -2845.819,Z -55.937,A 89.97773,B 0.00000,C 180.00000} ; insert
  LIN {X 14031.817,Y -2845.819,Z -55.937,A 89.97773,B 0.00000,C 180.00000} ; release
  LIN {X 14031.817,Y -2845.819,Z 244.063,A 89.97773,B 0.00000,C 180.00000} ; retreat
  ; Step 2368, bar 611
  LIN {X -14031.817,Y 2845.819,Z 1147.317,A -90.02227,B 0.00000,C -180.00000} ; outside
  LIN {X -14031.817,Y 2845.819,Z 194.063,A -90.02227,B 0.00000,C -180.00000} ; preinsert
  LIN {X -14031.817,Y 2845.819,Z -55.937,A -90.02227,B 0.00000,C -180.00000} ; insert
  LIN {X -14031.817,Y 2845.819,Z -55.937,A -90.02227,B 0.00000,C -180.00000} ; release
  LIN {X -14031.817,Y 2845.819,Z 244.063,A -90.02227,B 0.00000,C -180.00000} ; retreat
  ; Step 2369, bar 609
  LIN {X -13931.817,Y 2845.819,Z 1147.317,A -90.02227,B 0.00000,C -180.00000} ; outside
  LIN {X -13931.817,Y 2845.819,Z 194.063,A -90.02227,B 0.00000,C -180.00000} ; preinsert
  LIN {X -13931.817,Y 2845.819,Z -55.937,A -90.02227,B 0.00000,C -180.00000} ; insert
  LIN {X -13931.817,Y 2845.819,Z -55.937,A -90.02227,B 0.00000,C -180.00000} ; release
  LIN {X -13931.817,Y 2845.819,Z 244.063,A -90.02227,B 0.00000,C -180.00000} ; retreat
  ; Step 2370, bar 615
  LIN {X -9981.817,Y 2845.819,Z 1147.317,A -90.02227,B 0.00000,C -180.00000} ; outside
  LIN {X -9981.817,Y 2845.819,Z 194.063,A -90.02227,B 0.00000,C -180.00000} ; preinsert
  LIN {X -9981.817,Y 2845.819,Z -55.937,A -90.02227,B 0.00000,C -180.00000} ; insert
  LIN {X -9981.817,Y 2845.819,Z -55.937,A -90.02227,B 0.00000,C -180.00000} ; release
  LIN {X -9981.817,Y 2845.819,Z 244.063,A -90.02227,B 0.00000,C -180.00000} ; retreat
  ; Step 2371, bar 613
  LIN {X -5981.817,Y 2845.819,Z 1147.317,A -90.02227,B 0.00000,C -180.00000} ; outside
  LIN {X -5981.817,Y 2845.819,Z 194.063,A -90.02227,B 0.00000,C -180.00000} ; preinsert
  LIN {X -5981.817,Y 2845.819,Z -55.937,A -90.02227,B 0.00000,C -180.00000} ; insert
  LIN {X -5981.817,Y 2845.819,Z -55.937,A -90.02227,B 0.00000,C -180.00000} ; release
  LIN {X -5981.817,Y 2845.819,Z 244.063,A -90.02227,B 0.00000,C -180.00000} ; retreat
  ; Step 2372, bar 617
  LIN {X -1981.817,Y 2845.819,Z 1147.317,A -90.02227,B 0.00000,C 180.00000} ; outside
  LIN {X -1981.817,Y 2845.819,Z 194.063,A -90.02227,B 0.00000,C 180.00000} ; preinsert
  LIN {X -1981.817,Y 2845.819,Z -55.937,A -90.02227,B 0.00000,C 180.00000} ; insert
  LIN {X -1981.817,Y 2845.819,Z -55.937,A -90.02227,B 0.00000,C 180.00000} ; release
  LIN {X -1981.817,Y 2845.819,Z 244.063,A -90.02227,B 0.00000,C 180.00000} ; retreat
  ; Step 2373, bar 1855
  LIN {X -14550.109,Y -1460.794,Z 819.651,A 90.04265,B 0.00000,C 180.00000} ; outside
  LIN {X -14550.109,Y -1460.794,Z -133.813,A 90.04265,B 0.00000,C 180.00000} ; preinsert
  LIN {X -14550.109,Y -1460.794,Z -383.813,A 90.04265,B 0.00000,C 180.00000} ; insert
  LIN {X -14550.109,Y -1460.794,Z -383.813,A 90.04265,B 0.00000,C 180.00000} ; release
  LIN {X -14550.109,Y -1460.794,Z -83.813,A 90.04265,B 0.00000,C 180.00000} ; retreat
  ; Step 2374, bar 1853
  LIN {X 14550.109,Y -1460.794,Z 819.651,A 89.95735,B 0.00000,C 180.00000} ; outside
  LIN {X 14550.109,Y -1460.794,Z -133.813,A 89.95735,B 0.00000,C 180.00000} ; preinsert
  LIN {X 14550.109,Y -1460.794,Z -383.813,A 89.95735,B 0.00000,C 180.00000} ; insert
  LIN {X 14550.109,Y -1460.794,Z -383.813,A 89.95735,B 0.00000,C 180.00000} ; release
  LIN {X 14550.109,Y -1460.794,Z -83.813,A 89.95735,B 0.00000,C 180.00000} ; retreat
  ; Step 2375, bar 2894
  LIN {X -11625.007,Y -731.780,Z 1072.618,A 90.84369,B 0.00000,C 180.00000} ; outside
  LIN {X -11625.007,Y -731.780,Z 116.320,A 90.84369,B 0.00000,C 180.00000} ; preinsert
  LIN {X -11625.007,Y -731.780,Z -133.680,A 90.84369,B 0.00000,C 180.00000} ; insert
  LIN {X -11625.007,Y -731.780,Z -133.680,A 90.84369,B 0.00000,C 180.00000} ; release
  LIN {X -11625.007,Y -731.780,Z 166.320,A 90.84369,B 0.00000,C 180.00000} ; retreat
  ; Step 2376, bar 2891
  LIN {X -10875.007,Y -731.780,Z 1072.618,A 90.84369,B 0.00000,C 180.00000} ; outside
  LIN {X -10875.007,Y -731.780,Z 116.320,A 90.84369,B 0.00000,C 180.00000} ; preinsert
  LIN {X -10875.007,Y -731.780,Z -133.680,A 90.84369,B 0.00000,C 180.00000} ; insert
  LIN {X -10875.007,Y -731.780,Z -133.680,A 90.84369,B 0.00000,C 180.00000} ; release
  LIN {X -10875.007,Y -731.780,Z 166.320,A 90.84369,B 0.00000,C 180.00000} ; retreat
  ; Step 2377, bar 2888
  LIN {X -10125.007,Y -731.780,Z 1072.618,A 90.84369,B 0.00000,C 180.00000} ; outside
  LIN {X -10125.007,Y -731.780,Z 116.320,A 90.84369,B 0.00000,C 180.00000} ; preinsert
  LIN {X -10125.007,Y -731.780,Z -133.680,A 90.84369,B 0.00000,C 180.00000} ; insert
  LIN {X -10125.007,Y -731.780,Z -133.680,A 90.84369,B 0.00000,C 180.00000} ; release
  LIN {X -10125.007,Y -731.780,Z 166.320,A 90.84369,B 0.00000,C 180.00000} ; retreat
  ; Step 2378, bar 2885
  LIN {X -9375.007,Y -731.780,Z 1072.618,A 90.84369,B 0.00000,C 180.00000} ; outside
  LIN {X -9375.007,Y -731.780,Z 116.320,A 90.84369,B 0.00000,C 180.00000} ; preinsert
  LIN {X -9375.007,Y -731.780,Z -133.680,A 90.84369,B 0.00000,C 180.00000} ; insert
  LIN {X -9375.007,Y -731.780,Z -133.680,A 90.84369,B 0.00000,C 180.00000} ; release
  LIN {X -9375.007,Y -731.780,Z 166.320,A 90.84369,B 0.00000,C 180.00000} ; retreat
  ; Step 2379, bar 2882
  LIN {X -8625.007,Y -731.780,Z 1072.618,A 90.84369,B 0.00000,C 180.00000} ; outside
  LIN {X -8625.007,Y -731.780,Z 116.320,A 90.84369,B 0.00000,C 180.00000} ; preinsert
  LIN {X -8625.007,Y -731.780,Z -133.680,A 90.84369,B 0.00000,C 180.00000} ; insert
  LIN {X -8625.007,Y -731.780,Z -133.680,A 90.84369,B 0.00000,C 180.00000} ; release
  LIN {X -8625.007,Y -731.780,Z 166.320,A 90.84369,B 0.00000,C 180.00000} ; retreat
  ; Step 2380, bar 2879
  LIN {X -7875.007,Y -731.780,Z 1072.618,A 90.84369,B 0.00000,C 180.00000} ; outside
  LIN {X -7875.007,Y -731.780,Z 116.320,A 90.84369,B 0.00000,C 180.00000} ; preinsert
  LIN {X -7875.007,Y -731.780,Z -133.680,A 90.84369,B 0.00000,C 180.00000} ; insert
  LIN {X -7875.007,Y -731.780,Z -133.680,A 90.84369,B 0.00000,C 180.00000} ; release
  LIN {X -7875.007,Y -731.780,Z 166.320,A 90.84369,B 0.00000,C 180.00000} ; retreat
  ; Step 2381, bar 2876
  LIN {X -7125.007,Y -731.780,Z 1072.618,A 90.84369,B 0.00000,C 180.00000} ; outside
  LIN {X -7125.007,Y -731.780,Z 116.320,A 90.84369,B 0.00000,C 180.00000} ; preinsert
  LIN {X -7125.007,Y -731.780,Z -133.680,A 90.84369,B 0.00000,C 180.00000} ; insert
  LIN {X -7125.007,Y -731.780,Z -133.680,A 90.84369,B 0.00000,C 180.00000} ; release
  LIN {X -7125.007,Y -731.780,Z 166.320,A 90.84369,B 0.00000,C 180.00000} ; retreat
  ; Step 2382, bar 2873
  LIN {X -6375.007,Y -731.780,Z 1072.618,A 90.84369,B 0.00000,C 180.00000} ; outside
  LIN {X -6375.007,Y -731.780,Z 116.320,A 90.84369,B 0.00000,C 180.00000} ; preinsert
  LIN {X -6375.007,Y -731.780,Z -133.680,A 90.84369,B 0.00000,C 180.00000} ; insert
  LIN {X -6375.007,Y -731.780,Z -133.680,A 90.84369,B 0.00000,C 180.00000} ; release
  LIN {X -6375.007,Y -731.780,Z 166.320,A 90.84369,B 0.00000,C 180.00000} ; retreat
  ; Step 2383, bar 2870
  LIN {X -5625.007,Y -731.780,Z 1072.618,A 90.84369,B 0.00000,C 180.00000} ; outside
  LIN {X -5625.007,Y -731.780,Z 116.320,A 90.84369,B 0.00000,C 180.00000} ; preinsert
  LIN {X -5625.007,Y -731.780,Z -133.680,A 90.84369,B 0.00000,C 180.00000} ; insert
  LIN {X -5625.007,Y -731.780,Z -133.680,A 90.84369,B 0.00000,C 180.00000} ; release
  LIN {X -5625.007,Y -731.780,Z 166.320,A 90.84369,B 0.00000,C 180.00000} ; retreat
  ; Step 2384, bar 2867
  LIN {X -4875.007,Y -731.780,Z 1072.618,A 90.84369,B 0.00000,C 180.00000} ; outside
  LIN {X -4875.007,Y -731.780,Z 116.320,A 90.84369,B 0.00000,C 180.00000} ; preinsert
  LIN {X -4875.007,Y -731.780,Z -133.680,A 90.84369,B 0.00000,C 180.00000} ; insert
  LIN {X -4875.007,Y -731.780,Z -133.680,A 90.84369,B 0.00000,C 180.00000} ; release
  LIN {X -4875.007,Y -731.780,Z 166.320,A 90.84369,B 0.00000,C 180.00000} ; retreat
  ; Step 2385, bar 2864
  LIN {X -4125.007,Y -731.780,Z 1072.618,A 90.84369,B 0.00000,C 180.00000} ; outside
  LIN {X -4125.007,Y -731.780,Z 116.320,A 90.84369,B 0.00000,C 180.00000} ; preinsert
  LIN {X -4125.007,Y -731.780,Z -133.680,A 90.84369,B 0.00000,C 180.00000} ; insert
  LIN {X -4125.007,Y -731.780,Z -133.680,A 90.84369,B 0.00000,C 180.00000} ; release
  LIN {X -4125.007,Y -731.780,Z 166.320,A 90.84369,B 0.00000,C 180.00000} ; retreat
  ; Step 2386, bar 2861
  LIN {X -3375.007,Y -731.780,Z 1072.618,A 90.84369,B 0.00000,C 180.00000} ; outside
  LIN {X -3375.007,Y -731.780,Z 116.320,A 90.84369,B 0.00000,C 180.00000} ; preinsert
  LIN {X -3375.007,Y -731.780,Z -133.680,A 90.84369,B 0.00000,C 180.00000} ; insert
  LIN {X -3375.007,Y -731.780,Z -133.680,A 90.84369,B 0.00000,C 180.00000} ; release
  LIN {X -3375.007,Y -731.780,Z 166.320,A 90.84369,B 0.00000,C 180.00000} ; retreat
  ; Step 2387, bar 2858
  LIN {X -2625.007,Y -731.780,Z 1072.618,A 90.84369,B 0.00000,C 180.00000} ; outside
  LIN {X -2625.007,Y -731.780,Z 116.320,A 90.84369,B 0.00000,C 180.00000} ; preinsert
  LIN {X -2625.007,Y -731.780,Z -133.680,A 90.84369,B 0.00000,C 180.00000} ; insert
  LIN {X -2625.007,Y -731.780,Z -133.680,A 90.84369,B 0.00000,C 180.00000} ; release
  LIN {X -2625.007,Y -731.780,Z 166.320,A 90.84369,B 0.00000,C 180.00000} ; retreat
  ; Step 2388, bar 2855
  LIN {X -1875.007,Y -731.780,Z 1072.618,A 90.84369,B 0.00000,C 180.00000} ; outside
  LIN {X -1875.007,Y -731.780,Z 116.320,A 90.84369,B 0.00000,C 180.00000} ; preinsert
  LIN {X -1875.007,Y -731.780,Z -133.680,A 90.84369,B 0.00000,C 180.00000} ; insert
  LIN {X -1875.007,Y -731.780,Z -133.680,A 90.84369,B 0.00000,C 180.00000} ; release
  LIN {X -1875.007,Y -731.780,Z 166.320,A 90.84369,B 0.00000,C 180.00000} ; retreat
  ; Step 2389, bar 2852
  LIN {X -1125.007,Y -731.780,Z 1072.618,A 90.84369,B 0.00000,C 180.00000} ; outside
  LIN {X -1125.007,Y -731.780,Z 116.320,A 90.84369,B 0.00000,C 180.00000} ; preinsert
  LIN {X -1125.007,Y -731.780,Z -133.680,A 90.84369,B 0.00000,C 180.00000} ; insert
  LIN {X -1125.007,Y -731.780,Z -133.680,A 90.84369,B 0.00000,C 180.00000} ; release
  LIN {X -1125.007,Y -731.780,Z 166.320,A 90.84369,B 0.00000,C 180.00000} ; retreat
  ; Step 2390, bar 2849
  LIN {X -375.007,Y -731.780,Z 1072.618,A 90.84369,B 0.00000,C 180.00000} ; outside
  LIN {X -375.007,Y -731.780,Z 116.320,A 90.84369,B 0.00000,C 180.00000} ; preinsert
  LIN {X -375.007,Y -731.780,Z -133.680,A 90.84369,B 0.00000,C 180.00000} ; insert
  LIN {X -375.007,Y -731.780,Z -133.680,A 90.84369,B 0.00000,C 180.00000} ; release
  LIN {X -375.007,Y -731.780,Z 166.320,A 90.84369,B 0.00000,C 180.00000} ; retreat
  ; Step 2391, bar 2897
  LIN {X 375.007,Y -731.780,Z 1072.618,A 89.15631,B 0.00000,C 180.00000} ; outside
  LIN {X 375.007,Y -731.780,Z 116.320,A 89.15631,B 0.00000,C 180.00000} ; preinsert
  LIN {X 375.007,Y -731.780,Z -133.680,A 89.15631,B 0.00000,C 180.00000} ; insert
  LIN {X 375.007,Y -731.780,Z -133.680,A 89.15631,B 0.00000,C 180.00000} ; release
  LIN {X 375.007,Y -731.780,Z 166.320,A 89.15631,B 0.00000,C 180.00000} ; retreat
  ; Step 2392, bar 2900
  LIN {X 1125.007,Y -731.780,Z 1072.618,A 89.15631,B 0.00000,C 180.00000} ; outside
  LIN {X 1125.007,Y -731.780,Z 116.320,A 89.15631,B 0.00000,C 180.00000} ; preinsert
  LIN {X 1125.007,Y -731.780,Z -133.680,A 89.15631,B 0.00000,C 180.00000} ; insert
  LIN {X 1125.007,Y -731.780,Z -133.680,A 89.15631,B 0.00000,C 180.00000} ; release
  LIN {X 1125.007,Y -731.780,Z 166.320,A 89.15631,B 0.00000,C 180.00000} ; retreat
  ; Step 2393, bar 2903
  LIN {X 1875.007,Y -731.780,Z 1072.618,A 89.15631,B 0.00000,C 180.00000} ; outside
  LIN {X 1875.007,Y -731.780,Z 116.320,A 89.15631,B 0.00000,C 180.00000} ; preinsert
  LIN {X 1875.007,Y -731.780,Z -133.680,A 89.15631,B 0.00000,C 180.00000} ; insert
  LIN {X 1875.007,Y -731.780,Z -133.680,A 89.15631,B 0.00000,C 180.00000} ; release
  LIN {X 1875.007,Y -731.780,Z 166.320,A 89.15631,B 0.00000,C 180.00000} ; retreat
  ; Step 2394, bar 2906
  LIN {X 2625.007,Y -731.780,Z 1072.618,A 89.15631,B 0.00000,C 180.00000} ; outside
  LIN {X 2625.007,Y -731.780,Z 116.320,A 89.15631,B 0.00000,C 180.00000} ; preinsert
  LIN {X 2625.007,Y -731.780,Z -133.680,A 89.15631,B 0.00000,C 180.00000} ; insert
  LIN {X 2625.007,Y -731.780,Z -133.680,A 89.15631,B 0.00000,C 180.00000} ; release
  LIN {X 2625.007,Y -731.780,Z 166.320,A 89.15631,B 0.00000,C 180.00000} ; retreat
  ; Step 2395, bar 2909
  LIN {X 3375.007,Y -731.780,Z 1072.618,A 89.15631,B 0.00000,C 180.00000} ; outside
  LIN {X 3375.007,Y -731.780,Z 116.320,A 89.15631,B 0.00000,C 180.00000} ; preinsert
  LIN {X 3375.007,Y -731.780,Z -133.680,A 89.15631,B 0.00000,C 180.00000} ; insert
  LIN {X 3375.007,Y -731.780,Z -133.680,A 89.15631,B 0.00000,C 180.00000} ; release
  LIN {X 3375.007,Y -731.780,Z 166.320,A 89.15631,B 0.00000,C 180.00000} ; retreat
  ; Step 2396, bar 2912
  LIN {X 4125.007,Y -731.780,Z 1072.618,A 89.15631,B 0.00000,C 180.00000} ; outside
  LIN {X 4125.007,Y -731.780,Z 116.320,A 89.15631,B 0.00000,C 180.00000} ; preinsert
  LIN {X 4125.007,Y -731.780,Z -133.680,A 89.15631,B 0.00000,C 180.00000} ; insert
  LIN {X 4125.007,Y -731.780,Z -133.680,A 89.15631,B 0.00000,C 180.00000} ; release
  LIN {X 4125.007,Y -731.780,Z 166.320,A 89.15631,B 0.00000,C 180.00000} ; retreat
  ; Step 2397, bar 2915
  LIN {X 4875.007,Y -731.780,Z 1072.618,A 89.15631,B 0.00000,C 180.00000} ; outside
  LIN {X 4875.007,Y -731.780,Z 116.320,A 89.15631,B 0.00000,C 180.00000} ; preinsert
  LIN {X 4875.007,Y -731.780,Z -133.680,A 89.15631,B 0.00000,C 180.00000} ; insert
  LIN {X 4875.007,Y -731.780,Z -133.680,A 89.15631,B 0.00000,C 180.00000} ; release
  LIN {X 4875.007,Y -731.780,Z 166.320,A 89.15631,B 0.00000,C 180.00000} ; retreat
  ; Step 2398, bar 2918
  LIN {X 5625.007,Y -731.780,Z 1072.618,A 89.15631,B 0.00000,C 180.00000} ; outside
  LIN {X 5625.007,Y -731.780,Z 116.320,A 89.15631,B 0.00000,C 180.00000} ; preinsert
  LIN {X 5625.007,Y -731.780,Z -133.680,A 89.15631,B 0.00000,C 180.00000} ; insert
  LIN {X 5625.007,Y -731.780,Z -133.680,A 89.15631,B 0.00000,C 180.00000} ; release
  LIN {X 5625.007,Y -731.780,Z 166.320,A 89.15631,B 0.00000,C 180.00000} ; retreat
  ; Step 2399, bar 2921
  LIN {X 6375.007,Y -731.780,Z 1072.618,A 89.15631,B 0.00000,C 180.00000} ; outside
  LIN {X 6375.007,Y -731.780,Z 116.320,A 89.15631,B 0.00000,C 180.00000} ; preinsert
  LIN {X 6375.007,Y -731.780,Z -133.680,A 89.15631,B 0.00000,C 180.00000} ; insert
  LIN {X 6375.007,Y -731.780,Z -133.680,A 89.15631,B 0.00000,C 180.00000} ; release
  LIN {X 6375.007,Y -731.780,Z 166.320,A 89.15631,B 0.00000,C 180.00000} ; retreat
  ; Step 2400, bar 2924
  LIN {X 7125.007,Y -731.780,Z 1072.618,A 89.15631,B 0.00000,C 180.00000} ; outside
  LIN {X 7125.007,Y -731.780,Z 116.320,A 89.15631,B 0.00000,C 180.00000} ; preinsert
  LIN {X 7125.007,Y -731.780,Z -133.680,A 89.15631,B 0.00000,C 180.00000} ; insert
  LIN {X 7125.007,Y -731.780,Z -133.680,A 89.15631,B 0.00000,C 180.00000} ; release
  LIN {X 7125.007,Y -731.780,Z 166.320,A 89.15631,B 0.00000,C 180.00000} ; retreat
  ; Step 2401, bar 2927
  LIN {X 7875.007,Y -731.780,Z 1072.618,A 89.15631,B 0.00000,C 180.00000} ; outside
  LIN {X 7875.007,Y -731.780,Z 116.320,A 89.15631,B 0.00000,C 180.00000} ; preinsert
  LIN {X 7875.007,Y -731.780,Z -133.680,A 89.15631,B 0.00000,C 180.00000} ; insert
  LIN {X 7875.007,Y -731.780,Z -133.680,A 89.15631,B 0.00000,C 180.00000} ; release
  LIN {X 7875.007,Y -731.780,Z 166.320,A 89.15631,B 0.00000,C 180.00000} ; retreat
  ; Step 2402, bar 2930
  LIN {X 8625.007,Y -731.780,Z 1072.618,A 89.15631,B 0.00000,C 180.00000} ; outside
  LIN {X 8625.007,Y -731.780,Z 116.320,A 89.15631,B 0.00000,C 180.00000} ; preinsert
  LIN {X 8625.007,Y -731.780,Z -133.680,A 89.15631,B 0.00000,C 180.00000} ; insert
  LIN {X 8625.007,Y -731.780,Z -133.680,A 89.15631,B 0.00000,C 180.00000} ; release
  LIN {X 8625.007,Y -731.780,Z 166.320,A 89.15631,B 0.00000,C 180.00000} ; retreat
  ; Step 2403, bar 2933
  LIN {X 9375.007,Y -731.780,Z 1072.618,A 89.15631,B 0.00000,C 180.00000} ; outside
  LIN {X 9375.007,Y -731.780,Z 116.320,A 89.15631,B 0.00000,C 180.00000} ; preinsert
  LIN {X 9375.007,Y -731.780,Z -133.680,A 89.15631,B 0.00000,C 180.00000} ; insert
  LIN {X 9375.007,Y -731.780,Z -133.680,A 89.15631,B 0.00000,C 180.00000} ; release
  LIN {X 9375.007,Y -731.780,Z 166.320,A 89.15631,B 0.00000,C 180.00000} ; retreat
  ; Step 2404, bar 2936
  LIN {X 10125.007,Y -731.780,Z 1072.618,A 89.15631,B 0.00000,C 180.00000} ; outside
  LIN {X 10125.007,Y -731.780,Z 116.320,A 89.15631,B 0.00000,C 180.00000} ; preinsert
  LIN {X 10125.007,Y -731.780,Z -133.680,A 89.15631,B 0.00000,C 180.00000} ; insert
  LIN {X 10125.007,Y -731.780,Z -133.680,A 89.15631,B 0.00000,C 180.00000} ; release
  LIN {X 10125.007,Y -731.780,Z 166.320,A 89.15631,B 0.00000,C 180.00000} ; retreat
  ; Step 2405, bar 2939
  LIN {X 10875.007,Y -731.780,Z 1072.618,A 89.15631,B 0.00000,C 180.00000} ; outside
  LIN {X 10875.007,Y -731.780,Z 116.320,A 89.15631,B 0.00000,C 180.00000} ; preinsert
  LIN {X 10875.007,Y -731.780,Z -133.680,A 89.15631,B 0.00000,C 180.00000} ; insert
  LIN {X 10875.007,Y -731.780,Z -133.680,A 89.15631,B 0.00000,C 180.00000} ; release
  LIN {X 10875.007,Y -731.780,Z 166.320,A 89.15631,B 0.00000,C 180.00000} ; retreat
  ; Step 2406, bar 2942
  LIN {X 11625.007,Y -731.780,Z 1072.618,A 89.15631,B 0.00000,C 180.00000} ; outside
  LIN {X 11625.007,Y -731.780,Z 116.320,A 89.15631,B 0.00000,C 180.00000} ; preinsert
  LIN {X 11625.007,Y -731.780,Z -133.680,A 89.15631,B 0.00000,C 180.00000} ; insert
  LIN {X 11625.007,Y -731.780,Z -133.680,A 89.15631,B 0.00000,C 180.00000} ; release
  LIN {X 11625.007,Y -731.780,Z 166.320,A 89.15631,B 0.00000,C 180.00000} ; retreat
  ; Step 2407, bar 2632
  LIN {X -11625.007,Y 731.780,Z 1072.618,A -90.84369,B 0.00000,C -180.00000} ; outside
  LIN {X -11625.007,Y 731.780,Z 116.320,A -90.84369,B 0.00000,C -180.00000} ; preinsert
  LIN {X -11625.007,Y 731.780,Z -133.680,A -90.84369,B 0.00000,C -180.00000} ; insert
  LIN {X -11625.007,Y 731.780,Z -133.680,A -90.84369,B 0.00000,C -180.00000} ; release
  LIN {X -11625.007,Y 731.780,Z 166.320,A -90.84369,B 0.00000,C -180.00000} ; retreat
  ; Step 2408, bar 2625
  LIN {X -10875.007,Y 731.780,Z 1072.618,A -90.84369,B 0.00000,C -180.00000} ; outside
  LIN {X -10875.007,Y 731.780,Z 116.320,A -90.84369,B 0.00000,C -180.00000} ; preinsert
  LIN {X -10875.007,Y 731.780,Z -133.680,A -90.84369,B 0.00000,C -180.00000} ; insert
  LIN {X -10875.007,Y 731.780,Z -133.680,A -90.84369,B 0.00000,C -180.00000} ; release
  LIN {X -10875.007,Y 731.780,Z 166.320,A -90.84369,B 0.00000,C -180.00000} ; retreat
  ; Step 2409, bar 2618
  LIN {X -10125.007,Y 731.780,Z 1072.618,A -90.84369,B 0.00000,C -180.00000} ; outside
  LIN {X -10125.007,Y 731.780,Z 116.320,A -90.84369,B 0.00000,C -180.00000} ; preinsert
  LIN {X -10125.007,Y 731.780,Z -133.680,A -90.84369,B 0.00000,C -180.00000} ; insert
  LIN {X -10125.007,Y 731.780,Z -133.680,A -90.84369,B 0.00000,C -180.00000} ; release
  LIN {X -10125.007,Y 731.780,Z 166.320,A -90.84369,B 0.00000,C -180.00000} ; retreat
  ; Step 2410, bar 2611
  LIN {X -9375.007,Y 731.780,Z 1072.618,A -90.84369,B 0.00000,C -180.00000} ; outside
  LIN {X -9375.007,Y 731.780,Z 116.320,A -90.84369,B 0.00000,C -180.00000} ; preinsert
  LIN {X -9375.007,Y 731.780,Z -133.680,A -90.84369,B 0.00000,C -180.00000} ; insert
  LIN {X -9375.007,Y 731.780,Z -133.680,A -90.84369,B 0.00000,C -180.00000} ; release
  LIN {X -9375.007,Y 731.780,Z 166.320,A -90.84369,B 0.00000,C -180.00000} ; retreat
  ; Step 2411, bar 2604
  LIN {X -8625.007,Y 731.780,Z 1072.618,A -90.84369,B 0.00000,C -180.00000} ; outside
  LIN {X -8625.007,Y 731.780,Z 116.320,A -90.84369,B 0.00000,C -180.00000} ; preinsert
  LIN {X -8625.007,Y 731.780,Z -133.680,A -90.84369,B 0.00000,C -180.00000} ; insert
  LIN {X -8625.007,Y 731.780,Z -133.680,A -90.84369,B 0.00000,C -180.00000} ; release
  LIN {X -8625.007,Y 731.780,Z 166.320,A -90.84369,B 0.00000,C -180.00000} ; retreat
  ; Step 2412, bar 2597
  LIN {X -7875.007,Y 731.780,Z 1072.618,A -90.84369,B 0.00000,C -180.00000} ; outside
  LIN {X -7875.007,Y 731.780,Z 116.320,A -90.84369,B 0.00000,C -180.00000} ; preinsert
  LIN {X -7875.007,Y 731.780,Z -133.680,A -90.84369,B 0.00000,C -180.00000} ; insert
  LIN {X -7875.007,Y 731.780,Z -133.680,A -90.84369,B 0.00000,C -180.00000} ; release
  LIN {X -7875.007,Y 731.780,Z 166.320,A -90.84369,B 0.00000,C -180.00000} ; retreat
  ; Step 2413, bar 2590
  LIN {X -7125.007,Y 731.780,Z 1072.618,A -90.84369,B 0.00000,C -180.00000} ; outside
  LIN {X -7125.007,Y 731.780,Z 116.320,A -90.84369,B 0.00000,C -180.00000} ; preinsert
  LIN {X -7125.007,Y 731.780,Z -133.680,A -90.84369,B 0.00000,C -180.00000} ; insert
  LIN {X -7125.007,Y 731.780,Z -133.680,A -90.84369,B 0.00000,C -180.00000} ; release
  LIN {X -7125.007,Y 731.780,Z 166.320,A -90.84369,B 0.00000,C -180.00000} ; retreat
  ; Step 2414, bar 2583
  LIN {X -6375.007,Y 731.780,Z 1072.618,A -90.84369,B 0.00000,C -180.00000} ; outside
  LIN {X -6375.007,Y 731.780,Z 116.320,A -90.84369,B 0.00000,C -180.00000} ; preinsert
  LIN {X -6375.007,Y 731.780,Z -133.680,A -90.84369,B 0.00000,C -180.00000} ; insert
  LIN {X -6375.007,Y 731.780,Z -133.680,A -90.84369,B 0.00000,C -180.00000} ; release
  LIN {X -6375.007,Y 731.780,Z 166.320,A -90.84369,B 0.00000,C -180.00000} ; retreat
  ; Step 2415, bar 2576
  LIN {X -5625.007,Y 731.780,Z 1072.618,A -90.84369,B 0.00000,C -180.00000} ; outside
  LIN {X -5625.007,Y 731.780,Z 116.320,A -90.84369,B 0.00000,C -180.00000} ; preinsert
  LIN {X -5625.007,Y 731.780,Z -133.680,A -90.84369,B 0.00000,C -180.00000} ; insert
  LIN {X -5625.007,Y 731.780,Z -133.680,A -90.84369,B 0.00000,C -180.00000} ; release
  LIN {X -5625.007,Y 731.780,Z 166.320,A -90.84369,B 0.00000,C -180.00000} ; retreat
  ; Step 2416, bar 2569
  LIN {X -4875.007,Y 731.780,Z 1072.618,A -90.84369,B 0.00000,C -180.00000} ; outside
  LIN {X -4875.007,Y 731.780,Z 116.320,A -90.84369,B 0.00000,C -180.00000} ; preinsert
  LIN {X -4875.007,Y 731.780,Z -133.680,A -90.84369,B 0.00000,C -180.00000} ; insert
  LIN {X -4875.007,Y 731.780,Z -133.680,A -90.84369,B 0.00000,C -180.00000} ; release
  LIN {X -4875.007,Y 731.780,Z 166.320,A -90.84369,B 0.00000,C -180.00000} ; retreat
  ; Step 2417, bar 2562
  LIN {X -4125.007,Y 731.780,Z 1072.618,A -90.84369,B 0.00000,C -180.00000} ; outside
  LIN {X -4125.007,Y 731.780,Z 116.320,A -90.84369,B 0.00000,C -180.00000} ; preinsert
  LIN {X -4125.007,Y 731.780,Z -133.680,A -90.84369,B 0.00000,C -180.00000} ; insert
  LIN {X -4125.007,Y 731.780,Z -133.680,A -90.84369,B 0.00000,C -180.00000} ; release
  LIN {X -4125.007,Y 731.780,Z 166.320,A -90.84369,B 0.00000,C -180.00000} ; retreat
  ; Step 2418, bar 2555
  LIN {X -3375.007,Y 731.780,Z 1072.618,A -90.84369,B 0.00000,C -180.00000} ; outside
  LIN {X -3375.007,Y 731.780,Z 116.320,A -90.84369,B 0.00000,C -180.00000} ; preinsert
  LIN {X -3375.007,Y 731.780,Z -133.680,A -90.84369,B 0.00000,C -180.00000} ; insert
  LIN {X -3375.007,Y 731.780,Z -133.680,A -90.84369,B 0.00000,C -180.00000} ; release
  LIN {X -3375.007,Y 731.780,Z 166.320,A -90.84369,B 0.00000,C -180.00000} ; retreat
  ; Step 2419, bar 2548
  LIN {X -2625.007,Y 731.780,Z 1072.618,A -90.84369,B 0.00000,C -180.00000} ; outside
  LIN {X -2625.007,Y 731.780,Z 116.320,A -90.84369,B 0.00000,C -180.00000} ; preinsert
  LIN {X -2625.007,Y 731.780,Z -133.680,A -90.84369,B 0.00000,C -180.00000} ; insert
  LIN {X -2625.007,Y 731.780,Z -133.680,A -90.84369,B 0.00000,C -180.00000} ; release
  LIN {X -2625.007,Y 731.780,Z 166.320,A -90.84369,B 0.00000,C -180.00000} ; retreat
  ; Step 2420, bar 2541
  LIN {X -1875.007,Y 731.780,Z 1072.618,A -90.84369,B 0.00000,C -180.00000} ; outside
  LIN {X -1875.007,Y 731.780,Z 116.320,A -90.84369,B 0.00000,C -180.00000} ; preinsert
  LIN {X -1875.007,Y 731.780,Z -133.680,A -90.84369,B 0.00000,C -180.00000} ; insert
  LIN {X -1875.007,Y 731.780,Z -133.680,A -90.84369,B 0.00000,C -180.00000} ; release
  LIN {X -1875.007,Y 731.780,Z 166.320,A -90.84369,B 0.00000,C -180.00000} ; retreat
  ; Step 2421, bar 2534
  LIN {X -1125.007,Y 731.780,Z 1072.618,A -90.84369,B 0.00000,C -180.00000} ; outside
  LIN {X -1125.007,Y 731.780,Z 116.320,A -90.84369,B 0.00000,C -180.00000} ; preinsert
  LIN {X -1125.007,Y 731.780,Z -133.680,A -90.84369,B 0.00000,C -180.00000} ; insert
  LIN {X -1125.007,Y 731.780,Z -133.680,A -90.84369,B 0.00000,C -180.00000} ; release
  LIN {X -1125.007,Y 731.780,Z 166.320,A -90.84369,B 0.00000,C -180.00000} ; retreat
  ; Step 2422, bar 1975
  LIN {X -375.007,Y 731.780,Z 1072.618,A -90.84369,B 0.00000,C -180.00000} ; outside
  LIN {X -375.007,Y 731.780,Z 116.320,A -90.84369,B 0.00000,C -180.00000} ; preinsert
  LIN {X -375.007,Y 731.780,Z -133.680,A -90.84369,B 0.00000,C -180.00000} ; insert
  LIN {X -375.007,Y 731.780,Z -133.680,A -90.84369,B 0.00000,C -180.00000} ; release
  LIN {X -375.007,Y 731.780,Z 166.320,A -90.84369,B 0.00000,C -180.00000} ; retreat
  ; Step 2423, bar 2686
  LIN {X 375.007,Y 731.780,Z 1072.618,A -89.15631,B 0.00000,C 180.00000} ; outside
  LIN {X 375.007,Y 731.780,Z 116.320,A -89.15631,B 0.00000,C 180.00000} ; preinsert
  LIN {X 375.007,Y 731.780,Z -133.680,A -89.15631,B 0.00000,C 180.00000} ; insert
  LIN {X 375.007,Y 731.780,Z -133.680,A -89.15631,B 0.00000,C 180.00000} ; release
  LIN {X 375.007,Y 731.780,Z 166.320,A -89.15631,B 0.00000,C 180.00000} ; retreat
  ; Step 2424, bar 2690
  LIN {X 1125.007,Y 731.780,Z 1072.618,A -89.15631,B 0.00000,C 180.00000} ; outside
  LIN {X 1125.007,Y 731.780,Z 116.320,A -89.15631,B 0.00000,C 180.00000} ; preinsert
  LIN {X 1125.007,Y 731.780,Z -133.680,A -89.15631,B 0.00000,C 180.00000} ; insert
  LIN {X 1125.007,Y 731.780,Z -133.680,A -89.15631,B 0.00000,C 180.00000} ; release
  LIN {X 1125.007,Y 731.780,Z 166.320,A -89.15631,B 0.00000,C 180.00000} ; retreat
  ; Step 2425, bar 2694
  LIN {X 1875.007,Y 731.780,Z 1072.618,A -89.15631,B 0.00000,C 180.00000} ; outside
  LIN {X 1875.007,Y 731.780,Z 116.320,A -89.15631,B 0.00000,C 180.00000} ; preinsert
  LIN {X 1875.007,Y 731.780,Z -133.680,A -89.15631,B 0.00000,C 180.00000} ; insert
  LIN {X 1875.007,Y 731.780,Z -133.680,A -89.15631,B 0.00000,C 180.00000} ; release
  LIN {X 1875.007,Y 731.780,Z 166.320,A -89.15631,B 0.00000,C 180.00000} ; retreat
  ; Step 2426, bar 2698
  LIN {X 2625.007,Y 731.780,Z 1072.618,A -89.15631,B 0.00000,C 180.00000} ; outside
  LIN {X 2625.007,Y 731.780,Z 116.320,A -89.15631,B 0.00000,C 180.00000} ; preinsert
  LIN {X 2625.007,Y 731.780,Z -133.680,A -89.15631,B 0.00000,C 180.00000} ; insert
  LIN {X 2625.007,Y 731.780,Z -133.680,A -89.15631,B 0.00000,C 180.00000} ; release
  LIN {X 2625.007,Y 731.780,Z 166.320,A -89.15631,B 0.00000,C 180.00000} ; retreat
  ; Step 2427, bar 2702
  LIN {X 3375.007,Y 731.780,Z 1072.618,A -89.15631,B 0.00000,C 180.00000} ; outside
  LIN {X 3375.007,Y 731.780,Z 116.320,A -89.15631,B 0.00000,C 180.00000} ; preinsert
  LIN {X 3375.007,Y 731.780,Z -133.680,A -89.15631,B 0.00000,C 180.00000} ; insert
  LIN {X 3375.007,Y 731.780,Z -133.680,A -89.15631,B 0.00000,C 180.00000} ; release
  LIN {X 3375.007,Y 731.780,Z 166.320,A -89.15631,B 0.00000,C 180.00000} ; retreat
  ; Step 2428, bar 2706
  LIN {X 4125.007,Y 731.780,Z 1072.618,A -89.15631,B 0.00000,C 180.00000} ; outside
  LIN {X 4125.007,Y 731.780,Z 116.320,A -89.15631,B 0.00000,C 180.00000} ; preinsert
  LIN {X 4125.007,Y 731.780,Z -133.680,A -89.15631,B 0.00000,C 180.00000} ; insert
  LIN {X 4125.007,Y 731.780,Z -133.680,A -89.15631,B 0.00000,C 180.00000} ; release
  LIN {X 4125.007,Y 731.780,Z 166.320,A -89.15631,B 0.00000,C 180.00000} ; retreat
  ; Step 2429, bar 2710
  LIN {X 4875.007,Y 731.780,Z 1072.618,A -89.15631,B 0.00000,C 180.00000} ; outside
  LIN {X 4875.007,Y 731.780,Z 116.320,A -89.15631,B 0.00000,C 180.00000} ; preinsert
  LIN {X 4875.007,Y 731.780,Z -133.680,A -89.15631,B 0.00000,C 180.00000} ; insert
  LIN {X 4875.007,Y 731.780,Z -133.680,A -89.15631,B 0.00000,C 180.00000} ; release
  LIN {X 4875.007,Y 731.780,Z 166.320,A -89.15631,B 0.00000,C 180.00000} ; retreat
  ; Step 2430, bar 2714
  LIN {X 5625.007,Y 731.780,Z 1072.618,A -89.15631,B 0.00000,C 180.00000} ; outside
  LIN {X 5625.007,Y 731.780,Z 116.320,A -89.15631,B 0.00000,C 180.00000} ; preinsert
  LIN {X 5625.007,Y 731.780,Z -133.680,A -89.15631,B 0.00000,C 180.00000} ; insert
  LIN {X 5625.007,Y 731.780,Z -133.680,A -89.15631,B 0.00000,C 180.00000} ; release
  LIN {X 5625.007,Y 731.780,Z 166.320,A -89.15631,B 0.00000,C 180.00000} ; retreat
  ; Step 2431, bar 2718
  LIN {X 6375.007,Y 731.780,Z 1072.618,A -89.15631,B 0.00000,C 180.00000} ; outside
  LIN {X 6375.007,Y 731.780,Z 116.320,A -89.15631,B 0.00000,C 180.00000} ; preinsert
  LIN {X 6375.007,Y 731.780,Z -133.680,A -89.15631,B 0.00000,C 180.00000} ; insert
  LIN {X 6375.007,Y 731.780,Z -133.680,A -89.15631,B 0.00000,C 180.00000} ; release
  LIN {X 6375.007,Y 731.780,Z 166.320,A -89.15631,B 0.00000,C 180.00000} ; retreat
  ; Step 2432, bar 2722
  LIN {X 7125.007,Y 731.780,Z 1072.618,A -89.15631,B 0.00000,C 180.00000} ; outside
  LIN {X 7125.007,Y 731.780,Z 116.320,A -89.15631,B 0.00000,C 180.00000} ; preinsert
  LIN {X 7125.007,Y 731.780,Z -133.680,A -89.15631,B 0.00000,C 180.00000} ; insert
  LIN {X 7125.007,Y 731.780,Z -133.680,A -89.15631,B 0.00000,C 180.00000} ; release
  LIN {X 7125.007,Y 731.780,Z 166.320,A -89.15631,B 0.00000,C 180.00000} ; retreat
  ; Step 2433, bar 2726
  LIN {X 7875.007,Y 731.780,Z 1072.618,A -89.15631,B 0.00000,C 180.00000} ; outside
  LIN {X 7875.007,Y 731.780,Z 116.320,A -89.15631,B 0.00000,C 180.00000} ; preinsert
  LIN {X 7875.007,Y 731.780,Z -133.680,A -89.15631,B 0.00000,C 180.00000} ; insert
  LIN {X 7875.007,Y 731.780,Z -133.680,A -89.15631,B 0.00000,C 180.00000} ; release
  LIN {X 7875.007,Y 731.780,Z 166.320,A -89.15631,B 0.00000,C 180.00000} ; retreat
  ; Step 2434, bar 2730
  LIN {X 8625.007,Y 731.780,Z 1072.618,A -89.15631,B 0.00000,C 180.00000} ; outside
  LIN {X 8625.007,Y 731.780,Z 116.320,A -89.15631,B 0.00000,C 180.00000} ; preinsert
  LIN {X 8625.007,Y 731.780,Z -133.680,A -89.15631,B 0.00000,C 180.00000} ; insert
  LIN {X 8625.007,Y 731.780,Z -133.680,A -89.15631,B 0.00000,C 180.00000} ; release
  LIN {X 8625.007,Y 731.780,Z 166.320,A -89.15631,B 0.00000,C 180.00000} ; retreat
  ; Step 2435, bar 2734
  LIN {X 9375.007,Y 731.780,Z 1072.618,A -89.15631,B 0.00000,C 180.00000} ; outside
  LIN {X 9375.007,Y 731.780,Z 116.320,A -89.15631,B 0.00000,C 180.00000} ; preinsert
  LIN {X 9375.007,Y 731.780,Z -133.680,A -89.15631,B 0.00000,C 180.00000} ; insert
  LIN {X 9375.007,Y 731.780,Z -133.680,A -89.15631,B 0.00000,C 180.00000} ; release
  LIN {X 9375.007,Y 731.780,Z 166.320,A -89.15631,B 0.00000,C 180.00000} ; retreat
  ; Step 2436, bar 2738
  LIN {X 10125.007,Y 731.780,Z 1072.618,A -89.15631,B 0.00000,C 180.00000} ; outside
  LIN {X 10125.007,Y 731.780,Z 116.320,A -89.15631,B 0.00000,C 180.00000} ; preinsert
  LIN {X 10125.007,Y 731.780,Z -133.680,A -89.15631,B 0.00000,C 180.00000} ; insert
  LIN {X 10125.007,Y 731.780,Z -133.680,A -89.15631,B 0.00000,C 180.00000} ; release
  LIN {X 10125.007,Y 731.780,Z 166.320,A -89.15631,B 0.00000,C 180.00000} ; retreat
  ; Step 2437, bar 2742
  LIN {X 10875.007,Y 731.780,Z 1072.618,A -89.15631,B 0.00000,C 180.00000} ; outside
  LIN {X 10875.007,Y 731.780,Z 116.320,A -89.15631,B 0.00000,C 180.00000} ; preinsert
  LIN {X 10875.007,Y 731.780,Z -133.680,A -89.15631,B 0.00000,C 180.00000} ; insert
  LIN {X 10875.007,Y 731.780,Z -133.680,A -89.15631,B 0.00000,C 180.00000} ; release
  LIN {X 10875.007,Y 731.780,Z 166.320,A -89.15631,B 0.00000,C 180.00000} ; retreat
  ; Step 2438, bar 2746
  LIN {X 11625.007,Y 731.780,Z 1072.618,A -89.15631,B 0.00000,C 180.00000} ; outside
  LIN {X 11625.007,Y 731.780,Z 116.320,A -89.15631,B 0.00000,C 180.00000} ; preinsert
  LIN {X 11625.007,Y 731.780,Z -133.680,A -89.15631,B 0.00000,C 180.00000} ; insert
  LIN {X 11625.007,Y 731.780,Z -133.680,A -89.15631,B 0.00000,C 180.00000} ; release
  LIN {X 11625.007,Y 731.780,Z 166.320,A -89.15631,B 0.00000,C 180.00000} ; retreat
  ; Step 2439, bar 2851
  LIN {X -749.916,Y -481.788,Z 1074.491,A 87.44234,B 0.00000,C 180.00000} ; outside
  LIN {X -749.916,Y -481.788,Z 116.006,A 87.44234,B 0.00000,C 180.00000} ; preinsert
  LIN {X -749.916,Y -481.788,Z -133.994,A 87.44234,B 0.00000,C 180.00000} ; insert
  LIN {X -749.916,Y -481.788,Z -133.994,A 87.44234,B 0.00000,C 180.00000} ; release
  LIN {X -749.916,Y -481.788,Z 166.006,A 87.44234,B 0.00000,C 180.00000} ; retreat
  ; Step 2440, bar 2899
  LIN {X 749.916,Y -481.788,Z 1074.491,A 92.55766,B 0.00000,C 180.00000} ; outside
  LIN {X 749.916,Y -481.788,Z 116.006,A 92.55766,B 0.00000,C 180.00000} ; preinsert
  LIN {X 749.916,Y -481.788,Z -133.994,A 92.55766,B 0.00000,C 180.00000} ; insert
  LIN {X 749.916,Y -481.788,Z -133.994,A 92.55766,B 0.00000,C 180.00000} ; release
  LIN {X 749.916,Y -481.788,Z 166.006,A 92.55766,B 0.00000,C 180.00000} ; retreat
  ; Step 2441, bar 2895
  LIN {X -11999.916,Y -481.788,Z 1074.491,A 87.44234,B 0.00000,C 180.00000} ; outside
  LIN {X -11999.916,Y -481.788,Z 116.006,A 87.44234,B 0.00000,C 180.00000} ; preinsert
  LIN {X -11999.916,Y -481.788,Z -133.994,A 87.44234,B 0.00000,C 180.00000} ; insert
  LIN {X -11999.916,Y -481.788,Z -133.994,A 87.44234,B 0.00000,C 180.00000} ; release
  LIN {X -11999.916,Y -481.788,Z 166.006,A 87.44234,B 0.00000,C 180.00000} ; retreat
  ; Step 2442, bar 2893
  LIN {X -11249.916,Y -481.788,Z 1074.491,A 87.44234,B 0.00000,C 180.00000} ; outside
  LIN {X -11249.916,Y -481.788,Z 116.006,A 87.44234,B 0.00000,C 180.00000} ; preinsert
  LIN {X -11249.916,Y -481.788,Z -133.994,A 87.44234,B 0.00000,C 180.00000} ; insert
  LIN {X -11249.916,Y -481.788,Z -133.994,A 87.44234,B 0.00000,C 180.00000} ; release
  LIN {X -11249.916,Y -481.788,Z 166.006,A 87.44234,B 0.00000,C 180.00000} ; retreat
  ; Step 2443, bar 2890
  LIN {X -10499.916,Y -481.788,Z 1074.491,A 87.44234,B 0.00000,C 180.00000} ; outside
  LIN {X -10499.916,Y -481.788,Z 116.006,A 87.44234,B 0.00000,C 180.00000} ; preinsert
  LIN {X -10499.916,Y -481.788,Z -133.994,A 87.44234,B 0.00000,C 180.00000} ; insert
  LIN {X -10499.916,Y -481.788,Z -133.994,A 87.44234,B 0.00000,C 180.00000} ; release
  LIN {X -10499.916,Y -481.788,Z 166.006,A 87.44234,B 0.00000,C 180.00000} ; retreat
  ; Step 2444, bar 2887
  LIN {X -9749.916,Y -481.788,Z 1074.491,A 87.44234,B 0.00000,C 180.00000} ; outside
  LIN {X -9749.916,Y -481.788,Z 116.006,A 87.44234,B 0.00000,C 180.00000} ; preinsert
  LIN {X -9749.916,Y -481.788,Z -133.994,A 87.44234,B 0.00000,C 180.00000} ; insert
  LIN {X -9749.916,Y -481.788,Z -133.994,A 87.44234,B 0.00000,C 180.00000} ; release
  LIN {X -9749.916,Y -481.788,Z 166.006,A 87.44234,B 0.00000,C 180.00000} ; retreat
  ; Step 2445, bar 2884
  LIN {X -8999.916,Y -481.788,Z 1074.491,A 87.44234,B 0.00000,C 180.00000} ; outside
  LIN {X -8999.916,Y -481.788,Z 116.006,A 87.44234,B 0.00000,C 180.00000} ; preinsert
  LIN {X -8999.916,Y -481.788,Z -133.994,A 87.44234,B 0.00000,C 180.00000} ; insert
  LIN {X -8999.916,Y -481.788,Z -133.994,A 87.44234,B 0.00000,C 180.00000} ; release
  LIN {X -8999.916,Y -481.788,Z 166.006,A 87.44234,B 0.00000,C 180.00000} ; retreat
  ; Step 2446, bar 2881
  LIN {X -8249.916,Y -481.788,Z 1074.491,A 87.44234,B 0.00000,C 180.00000} ; outside
  LIN {X -8249.916,Y -481.788,Z 116.006,A 87.44234,B 0.00000,C 180.00000} ; preinsert
  LIN {X -8249.916,Y -481.788,Z -133.994,A 87.44234,B 0.00000,C 180.00000} ; insert
  LIN {X -8249.916,Y -481.788,Z -133.994,A 87.44234,B 0.00000,C 180.00000} ; release
  LIN {X -8249.916,Y -481.788,Z 166.006,A 87.44234,B 0.00000,C 180.00000} ; retreat
  ; Step 2447, bar 2878
  LIN {X -7499.916,Y -481.788,Z 1074.491,A 87.44234,B 0.00000,C 180.00000} ; outside
  LIN {X -7499.916,Y -481.788,Z 116.006,A 87.44234,B 0.00000,C 180.00000} ; preinsert
  LIN {X -7499.916,Y -481.788,Z -133.994,A 87.44234,B 0.00000,C 180.00000} ; insert
  LIN {X -7499.916,Y -481.788,Z -133.994,A 87.44234,B 0.00000,C 180.00000} ; release
  LIN {X -7499.916,Y -481.788,Z 166.006,A 87.44234,B 0.00000,C 180.00000} ; retreat
  ; Step 2448, bar 2875
  LIN {X -6749.916,Y -481.788,Z 1074.491,A 87.44234,B 0.00000,C 180.00000} ; outside
  LIN {X -6749.916,Y -481.788,Z 116.006,A 87.44234,B 0.00000,C 180.00000} ; preinsert
  LIN {X -6749.916,Y -481.788,Z -133.994,A 87.44234,B 0.00000,C 180.00000} ; insert
  LIN {X -6749.916,Y -481.788,Z -133.994,A 87.44234,B 0.00000,C 180.00000} ; release
  LIN {X -6749.916,Y -481.788,Z 166.006,A 87.44234,B 0.00000,C 180.00000} ; retreat
  ; Step 2449, bar 2872
  LIN {X -5999.916,Y -481.788,Z 1074.491,A 87.44234,B 0.00000,C 180.00000} ; outside
  LIN {X -5999.916,Y -481.788,Z 116.006,A 87.44234,B 0.00000,C 180.00000} ; preinsert
  LIN {X -5999.916,Y -481.788,Z -133.994,A 87.44234,B 0.00000,C 180.00000} ; insert
  LIN {X -5999.916,Y -481.788,Z -133.994,A 87.44234,B 0.00000,C 180.00000} ; release
  LIN {X -5999.916,Y -481.788,Z 166.006,A 87.44234,B 0.00000,C 180.00000} ; retreat
  ; Step 2450, bar 2869
  LIN {X -5249.916,Y -481.788,Z 1074.491,A 87.44234,B 0.00000,C 180.00000} ; outside
  LIN {X -5249.916,Y -481.788,Z 116.006,A 87.44234,B 0.00000,C 180.00000} ; preinsert
  LIN {X -5249.916,Y -481.788,Z -133.994,A 87.44234,B 0.00000,C 180.00000} ; insert
  LIN {X -5249.916,Y -481.788,Z -133.994,A 87.44234,B 0.00000,C 180.00000} ; release
  LIN {X -5249.916,Y -481.788,Z 166.006,A 87.44234,B 0.00000,C 180.00000} ; retreat
  ; Step 2451, bar 2866
  LIN {X -4499.916,Y -481.788,Z 1074.491,A 87.44234,B 0.00000,C 180.00000} ; outside
  LIN {X -4499.916,Y -481.788,Z 116.006,A 87.44234,B 0.00000,C 180.00000} ; preinsert
  LIN {X -4499.916,Y -481.788,Z -133.994,A 87.44234,B 0.00000,C 180.00000} ; insert
  LIN {X -4499.916,Y -481.788,Z -133.994,A 87.44234,B 0.00000,C 180.00000} ; release
  LIN {X -4499.916,Y -481.788,Z 166.006,A 87.44234,B 0.00000,C 180.00000} ; retreat
  ; Step 2452, bar 2863
  LIN {X -3749.916,Y -481.788,Z 1074.491,A 87.44234,B 0.00000,C 180.00000} ; outside
  LIN {X -3749.916,Y -481.788,Z 116.006,A 87.44234,B 0.00000,C 180.00000} ; preinsert
  LIN {X -3749.916,Y -481.788,Z -133.994,A 87.44234,B 0.00000,C 180.00000} ; insert
  LIN {X -3749.916,Y -481.788,Z -133.994,A 87.44234,B 0.00000,C 180.00000} ; release
  LIN {X -3749.916,Y -481.788,Z 166.006,A 87.44234,B 0.00000,C 180.00000} ; retreat
  ; Step 2453, bar 2860
  LIN {X -2999.916,Y -481.788,Z 1074.491,A 87.44234,B 0.00000,C 180.00000} ; outside
  LIN {X -2999.916,Y -481.788,Z 116.006,A 87.44234,B 0.00000,C 180.00000} ; preinsert
  LIN {X -2999.916,Y -481.788,Z -133.994,A 87.44234,B 0.00000,C 180.00000} ; insert
  LIN {X -2999.916,Y -481.788,Z -133.994,A 87.44234,B 0.00000,C 180.00000} ; release
  LIN {X -2999.916,Y -481.788,Z 166.006,A 87.44234,B 0.00000,C 180.00000} ; retreat
  ; Step 2454, bar 2857
  LIN {X -2249.916,Y -481.788,Z 1074.491,A 87.44234,B 0.00000,C 180.00000} ; outside
  LIN {X -2249.916,Y -481.788,Z 116.006,A 87.44234,B 0.00000,C 180.00000} ; preinsert
  LIN {X -2249.916,Y -481.788,Z -133.994,A 87.44234,B 0.00000,C 180.00000} ; insert
  LIN {X -2249.916,Y -481.788,Z -133.994,A 87.44234,B 0.00000,C 180.00000} ; release
  LIN {X -2249.916,Y -481.788,Z 166.006,A 87.44234,B 0.00000,C 180.00000} ; retreat
  ; Step 2455, bar 2854
  LIN {X -1499.916,Y -481.788,Z 1074.491,A 87.44234,B 0.00000,C 180.00000} ; outside
  LIN {X -1499.916,Y -481.788,Z 116.006,A 87.44234,B 0.00000,C 180.00000} ; preinsert
  LIN {X -1499.916,Y -481.788,Z -133.994,A 87.44234,B 0.00000,C 180.00000} ; insert
  LIN {X -1499.916,Y -481.788,Z -133.994,A 87.44234,B 0.00000,C 180.00000} ; release
  LIN {X -1499.916,Y -481.788,Z 166.006,A 87.44234,B 0.00000,C 180.00000} ; retreat
  ; Step 2456, bar 2848
  LIN {X 0.084,Y -481.788,Z 1074.491,A 87.44234,B 0.00000,C 180.00000} ; outside
  LIN {X 0.084,Y -481.788,Z 116.006,A 87.44234,B 0.00000,C 180.00000} ; preinsert
  LIN {X 0.084,Y -481.788,Z -133.994,A 87.44234,B 0.00000,C 180.00000} ; insert
  LIN {X 0.084,Y -481.788,Z -133.994,A 87.44234,B 0.00000,C 180.00000} ; release
  LIN {X 0.084,Y -481.788,Z 166.006,A 87.44234,B 0.00000,C 180.00000} ; retreat
  ; Step 2457, bar 2902
  LIN {X 1499.916,Y -481.788,Z 1074.491,A 92.55766,B 0.00000,C 180.00000} ; outside
  LIN {X 1499.916,Y -481.788,Z 116.006,A 92.55766,B 0.00000,C 180.00000} ; preinsert
